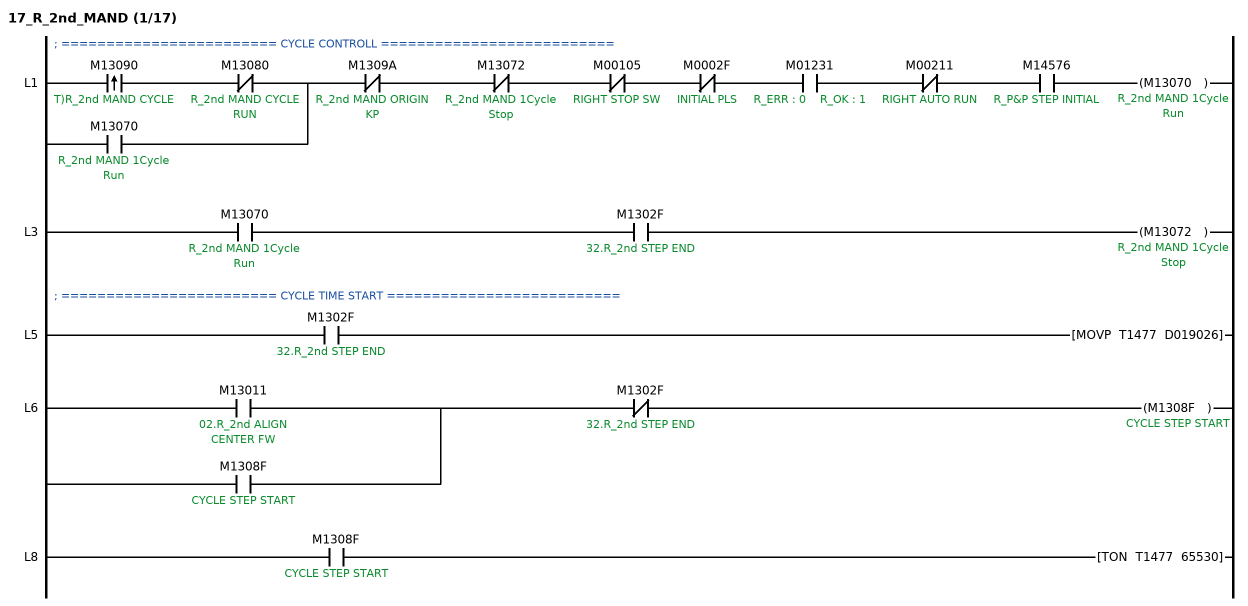
[picture p144: 17_R_2nd_MAND rungs L1-L8]
// ======================== CYCLE CONTROLL ==========================
; L1
LOADP     M13090	// T)R_2nd MAND CYCLE
AND NOT   M13080	// R_2nd MAND CYCLE RUN
OR        M13070	// R_2nd MAND 1Cycle Run
AND NOT   M1309A	// R_2nd MAND ORIGIN KP
AND NOT   M13072	// R_2nd MAND 1Cycle Stop
AND NOT   M00105	// RIGHT STOP SW
AND NOT   M0002F	// INITIAL PLS
AND       M01231	// R_ERR : 0    R_OK : 1
AND NOT   M00211	// RIGHT AUTO RUN
AND       M14576	// R_P&P STEP INITIAL
OUT       M13070	// R_2nd MAND 1Cycle Run
; L3
LOAD      M13070	// R_2nd MAND 1Cycle Run
AND       M1302F	// 32.R_2nd STEP END
OUT       M13072	// R_2nd MAND 1Cycle Stop
// ======================== CYCLE TIME START ==========================
; L5
LOAD      M1302F	// 32.R_2nd STEP END
MOVP      T1477 D019026
; L6
LOAD      M13011	// 02.R_2nd ALIGN CENTER FW
OR        M1308F	// CYCLE STEP START
AND NOT   M1302F	// 32.R_2nd STEP END
OUT       M1308F	// CYCLE STEP START
; L8
LOAD      M1308F	// CYCLE STEP START
TON       T1477 65530

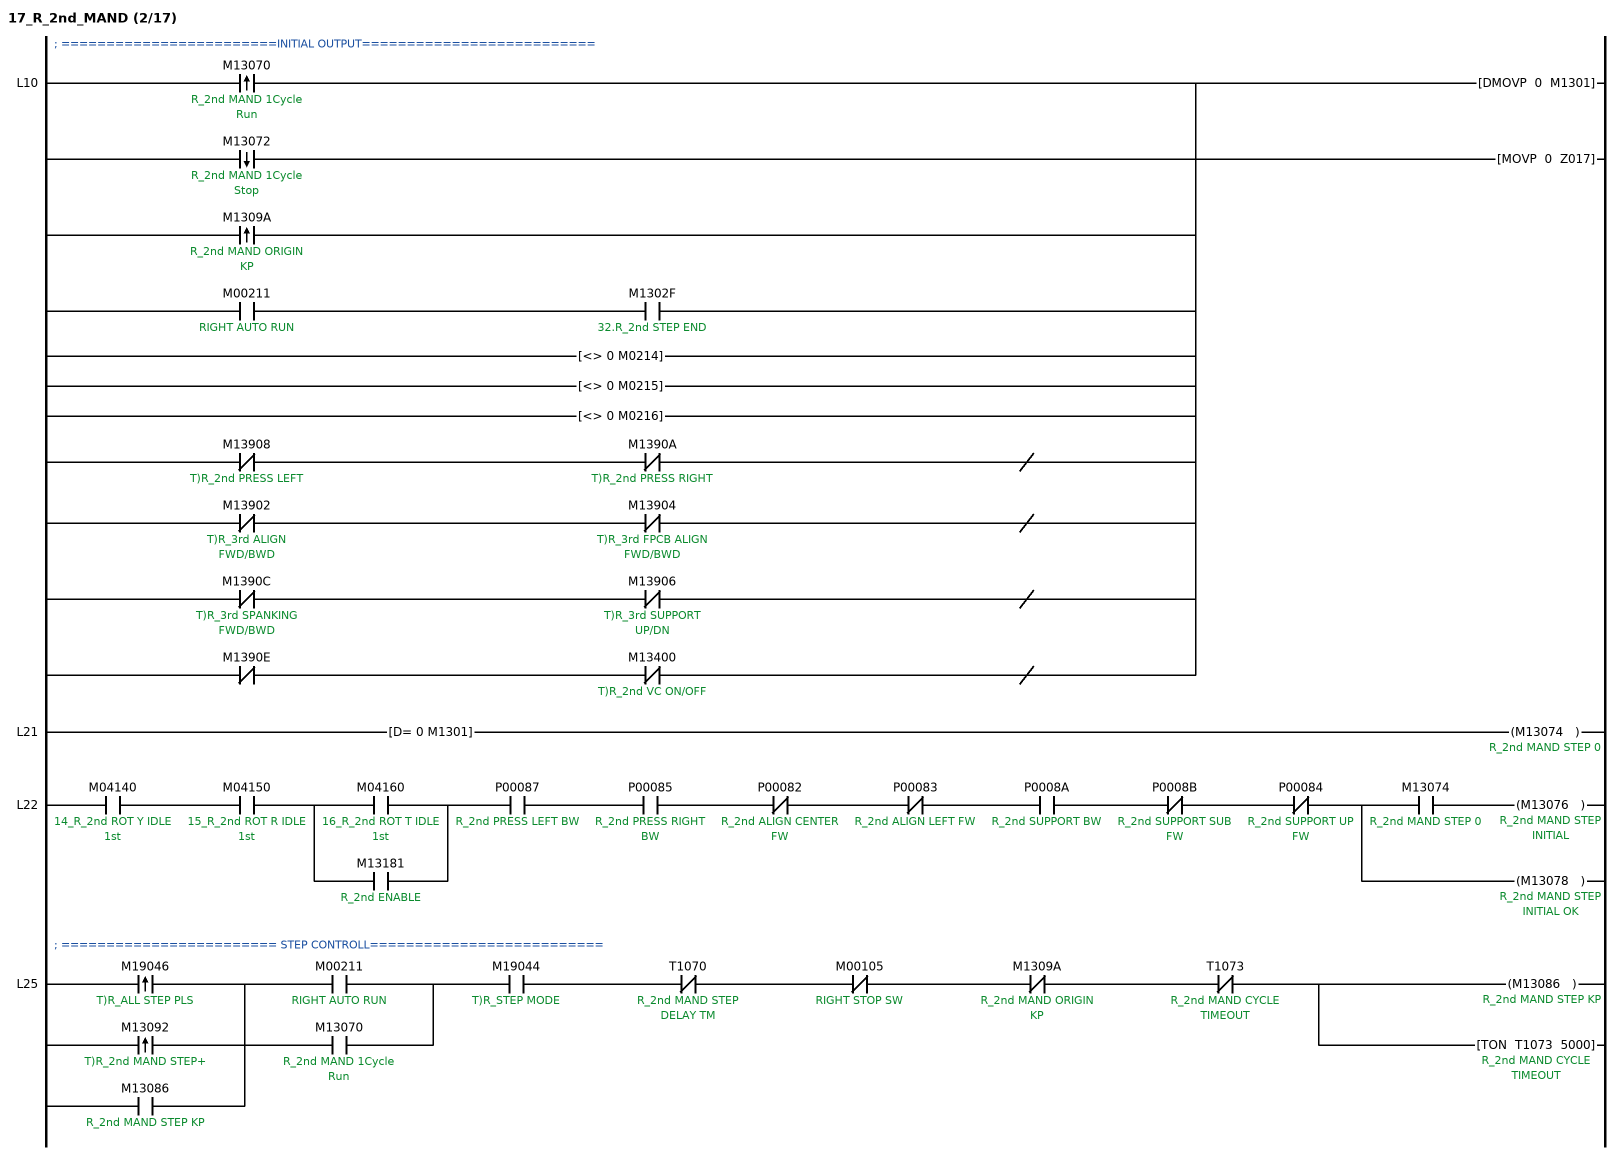
// ========================INITIAL OUTPUT==========================
; L10
LOADP     M13070	// R_2nd MAND 1Cycle Run
ORN       M13072	// R_2nd MAND 1Cycle Stop
ORP       M1309A	// R_2nd MAND ORIGIN KP
LOAD      M00211	// RIGHT AUTO RUN
AND       M1302F	// 32.R_2nd STEP END
OR LOAD
OR<>      0 M0214
OR<>      0 M0215
OR<>      0 M0216
LOAD NOT  M13908	// T)R_2nd PRESS LEFT
AND NOT   M1390A	// T)R_2nd PRESS RIGHT
NOT
OR LOAD
LOAD NOT  M13902	// T)R_3rd ALIGN FWD/BWD
AND NOT   M13904	// T)R_3rd FPCB ALIGN FWD/BWD
NOT
OR LOAD
LOAD NOT  M1390C	// T)R_3rd SPANKING FWD/BWD
AND NOT   M13906	// T)R_3rd SUPPORT UP/DN
NOT
OR LOAD
LOAD NOT  M1390E
AND NOT   M13400	// T)R_2nd VC ON/OFF
NOT
OR LOAD
DMOVP     0 M1301
MOVP      0 Z017
; L21
LOADD=    0 M1301
OUT       M13074	// R_2nd MAND STEP 0
; L22
LOAD      M04140	// 14_R_2nd ROT Y IDLE 1st
AND       M04150	// 15_R_2nd ROT R IDLE 1st
LOAD      M04160	// 16_R_2nd ROT T IDLE 1st
OR        M13181	// R_2nd ENABLE
AND LOAD
AND       P00087	// R_2nd PRESS LEFT BW
AND       P00085	// R_2nd PRESS RIGHT BW
AND NOT   P00082	// R_2nd ALIGN CENTER FW
AND NOT   P00083	// R_2nd ALIGN LEFT FW
AND       P0008A	// R_2nd SUPPORT BW
AND NOT   P0008B	// R_2nd SUPPORT SUB FW
AND NOT   P00084	// R_2nd SUPPORT UP FW
MPUSH
AND       M13074	// R_2nd MAND STEP 0
OUT       M13076	// R_2nd MAND STEP INITIAL
MPOP
OUT       M13078	// R_2nd MAND STEP INITIAL OK
// ======================== STEP CONTROLL==========================
; L25
LOADP     M19046	// T)R_ALL STEP PLS
ORP       M13092	// T)R_2nd MAND STEP+
OR        M13086	// R_2nd MAND STEP KP
LOAD      M00211	// RIGHT AUTO RUN
OR        M13070	// R_2nd MAND 1Cycle Run
AND LOAD
AND       M19044	// T)R_STEP MODE
AND NOT   T1070	// R_2nd MAND STEP DELAY TM
AND NOT   M00105	// RIGHT STOP SW
AND NOT   M1309A	// R_2nd MAND ORIGIN KP
AND NOT   T1073	// R_2nd MAND CYCLE TIMEOUT
OUT       M13086	// R_2nd MAND STEP KP
TON       T1073 5000	// R_2nd MAND CYCLE TIMEOUT

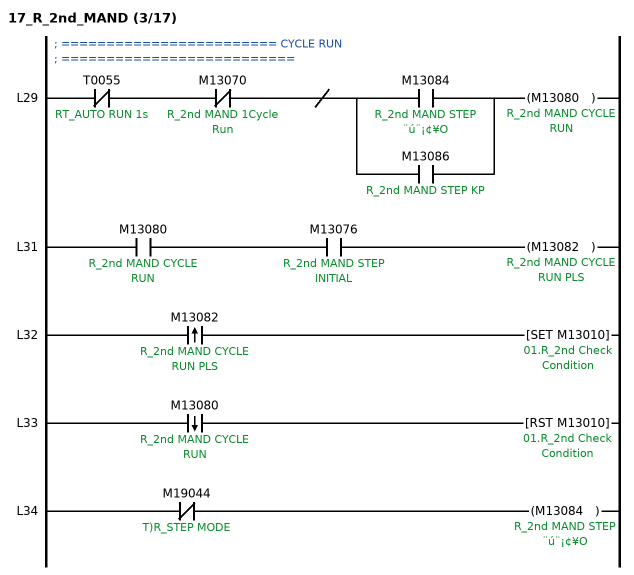
// ======================== CYCLE RUN ==========================
; L29
LOAD NOT  T0055	// RT_AUTO RUN 1s
AND NOT   M13070	// R_2nd MAND 1Cycle Run
NOT
LOAD      M13084	// R_2nd MAND STEP ¨ú¨¡¢¥O
OR        M13086	// R_2nd MAND STEP KP
AND LOAD
OUT       M13080	// R_2nd MAND CYCLE RUN
; L31
LOAD      M13080	// R_2nd MAND CYCLE RUN
AND       M13076	// R_2nd MAND STEP INITIAL
OUT       M13082	// R_2nd MAND CYCLE RUN PLS
; L32
LOADP     M13082	// R_2nd MAND CYCLE RUN PLS
SET       M13010	// 01.R_2nd Check Condition
; L33
LOADN     M13080	// R_2nd MAND CYCLE RUN
RST       M13010	// 01.R_2nd Check Condition
; L34
LOAD NOT  M19044	// T)R_STEP MODE
OUT       M13084	// R_2nd MAND STEP ¨ú¨¡¢¥O

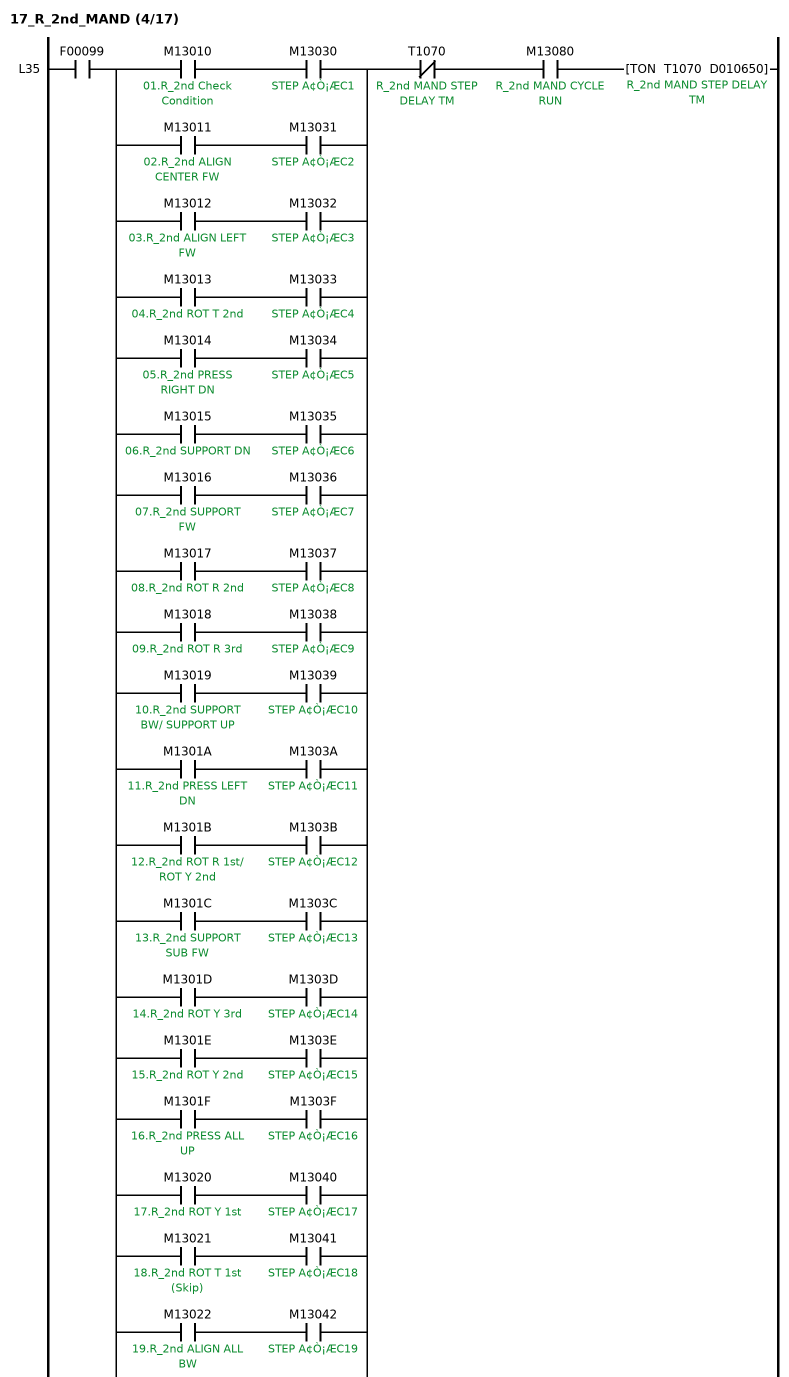

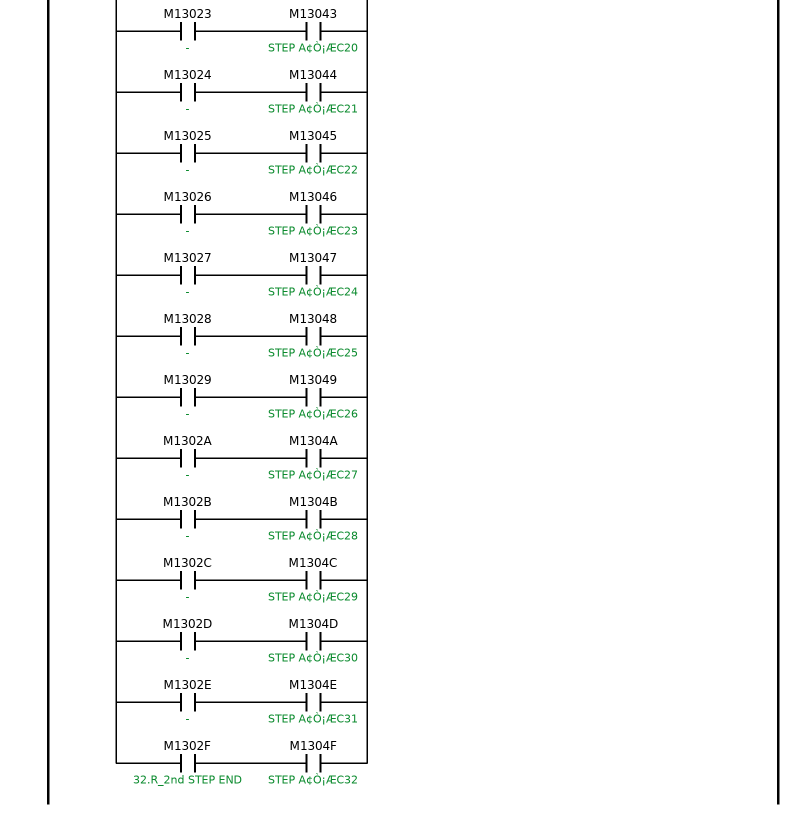
; L35
LOAD      F00099
LOAD      M13010	// 01.R_2nd Check Condition
AND       M13030	// STEP A¢Ò¡ÆC1
LOAD      M13011	// 02.R_2nd ALIGN CENTER FW
AND       M13031	// STEP A¢Ò¡ÆC2
OR LOAD
LOAD      M13012	// 03.R_2nd ALIGN LEFT FW
AND       M13032	// STEP A¢Ò¡ÆC3
OR LOAD
LOAD      M13013	// 04.R_2nd ROT T 2nd
AND       M13033	// STEP A¢Ò¡ÆC4
OR LOAD
LOAD      M13014	// 05.R_2nd PRESS RIGHT DN
AND       M13034	// STEP A¢Ò¡ÆC5
OR LOAD
LOAD      M13015	// 06.R_2nd SUPPORT DN
AND       M13035	// STEP A¢Ò¡ÆC6
OR LOAD
LOAD      M13016	// 07.R_2nd SUPPORT FW
AND       M13036	// STEP A¢Ò¡ÆC7
OR LOAD
LOAD      M13017	// 08.R_2nd ROT R 2nd
AND       M13037	// STEP A¢Ò¡ÆC8
OR LOAD
LOAD      M13018	// 09.R_2nd ROT R 3rd
AND       M13038	// STEP A¢Ò¡ÆC9
OR LOAD
LOAD      M13019	// 10.R_2nd SUPPORT BW/ SUPPORT UP
AND       M13039	// STEP A¢Ò¡ÆC10
OR LOAD
LOAD      M1301A	// 11.R_2nd PRESS LEFT DN
AND       M1303A	// STEP A¢Ò¡ÆC11
OR LOAD
LOAD      M1301B	// 12.R_2nd ROT R 1st/ ROT Y 2nd
AND       M1303B	// STEP A¢Ò¡ÆC12
OR LOAD
LOAD      M1301C	// 13.R_2nd SUPPORT SUB FW
AND       M1303C	// STEP A¢Ò¡ÆC13
OR LOAD
LOAD      M1301D	// 14.R_2nd ROT Y 3rd
AND       M1303D	// STEP A¢Ò¡ÆC14
OR LOAD
LOAD      M1301E	// 15.R_2nd ROT Y 2nd
AND       M1303E	// STEP A¢Ò¡ÆC15
OR LOAD
LOAD      M1301F	// 16.R_2nd PRESS ALL UP
AND       M1303F	// STEP A¢Ò¡ÆC16
OR LOAD
LOAD      M13020	// 17.R_2nd ROT Y 1st
AND       M13040	// STEP A¢Ò¡ÆC17
OR LOAD
LOAD      M13021	// 18.R_2nd ROT T 1st (Skip)
AND       M13041	// STEP A¢Ò¡ÆC18
OR LOAD
LOAD      M13022	// 19.R_2nd ALIGN ALL BW
AND       M13042	// STEP A¢Ò¡ÆC19
OR LOAD
LOAD      M13023	// -
AND       M13043	// STEP A¢Ò¡ÆC20
OR LOAD
LOAD      M13024	// -
AND       M13044	// STEP A¢Ò¡ÆC21
OR LOAD
LOAD      M13025	// -
AND       M13045	// STEP A¢Ò¡ÆC22
OR LOAD
LOAD      M13026	// -
AND       M13046	// STEP A¢Ò¡ÆC23
OR LOAD
LOAD      M13027	// -
AND       M13047	// STEP A¢Ò¡ÆC24
OR LOAD
LOAD      M13028	// -
AND       M13048	// STEP A¢Ò¡ÆC25
OR LOAD
LOAD      M13029	// -
AND       M13049	// STEP A¢Ò¡ÆC26
OR LOAD
LOAD      M1302A	// -
AND       M1304A	// STEP A¢Ò¡ÆC27
OR LOAD
LOAD      M1302B	// -
AND       M1304B	// STEP A¢Ò¡ÆC28
OR LOAD
LOAD      M1302C	// -
AND       M1304C	// STEP A¢Ò¡ÆC29
OR LOAD
LOAD      M1302D	// -
AND       M1304D	// STEP A¢Ò¡ÆC30
OR LOAD
LOAD      M1302E	// -
AND       M1304E	// STEP A¢Ò¡ÆC31
OR LOAD
LOAD      M1302F	// 32.R_2nd STEP END
AND       M1304F	// STEP A¢Ò¡ÆC32
OR LOAD
AND LOAD
AND NOT   T1070	// R_2nd MAND STEP DELAY TM
AND       M13080	// R_2nd MAND CYCLE RUN
TON       T1070 D010650	// R_2nd MAND STEP DELAY TM

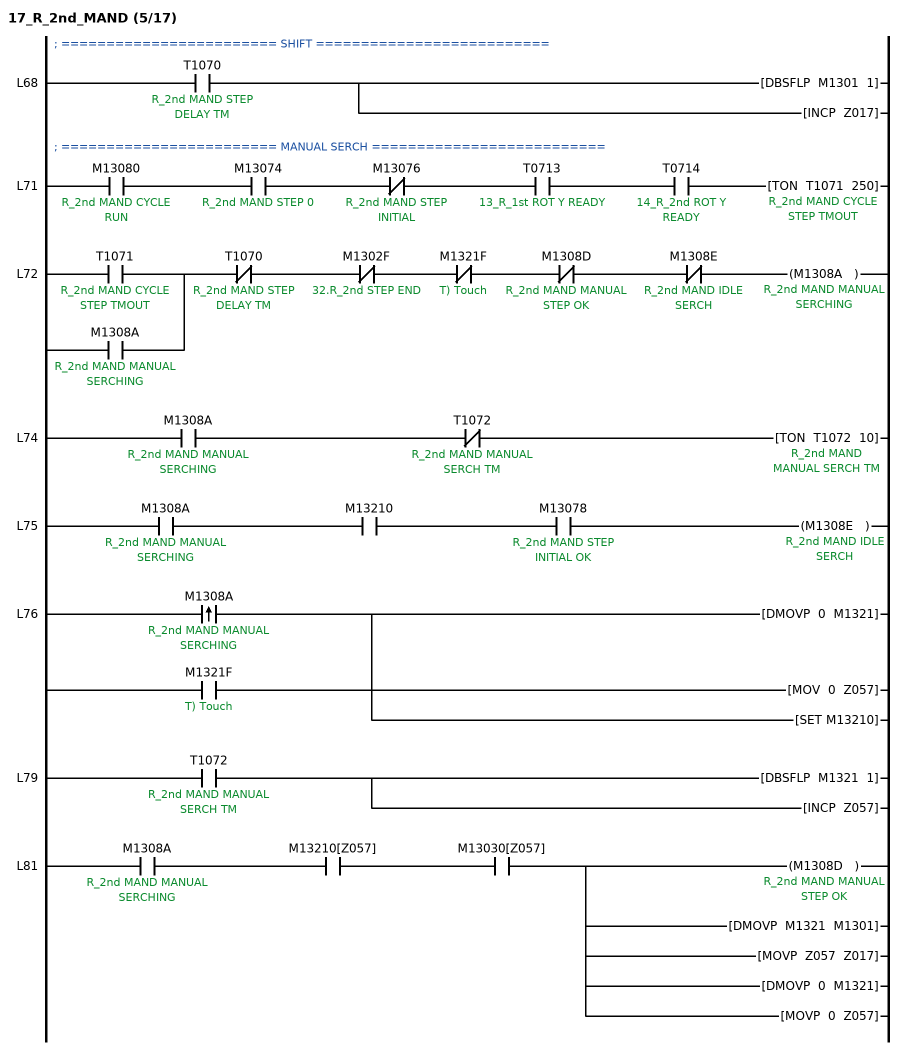
// ======================== SHIFT ==========================
; L68
LOAD      T1070	// R_2nd MAND STEP DELAY TM
DBSFLP    M1301 1
INCP      Z017
// ======================== MANUAL SERCH ==========================
; L71
LOAD      M13080	// R_2nd MAND CYCLE RUN
AND       M13074	// R_2nd MAND STEP 0
AND NOT   M13076	// R_2nd MAND STEP INITIAL
AND       T0713	// 13_R_1st ROT Y READY
AND       T0714	// 14_R_2nd ROT Y READY
TON       T1071 250	// R_2nd MAND CYCLE STEP TMOUT
; L72
LOAD      T1071	// R_2nd MAND CYCLE STEP TMOUT
OR        M1308A	// R_2nd MAND MANUAL SERCHING
AND NOT   T1070	// R_2nd MAND STEP DELAY TM
AND NOT   M1302F	// 32.R_2nd STEP END
AND NOT   M1321F	// T) Touch
AND NOT   M1308D	// R_2nd MAND MANUAL STEP OK
AND NOT   M1308E	// R_2nd MAND IDLE SERCH
OUT       M1308A	// R_2nd MAND MANUAL SERCHING
; L74
LOAD      M1308A	// R_2nd MAND MANUAL SERCHING
AND NOT   T1072	// R_2nd MAND MANUAL SERCH TM
TON       T1072 10	// R_2nd MAND MANUAL SERCH TM
; L75
LOAD      M1308A	// R_2nd MAND MANUAL SERCHING
AND       M13210
AND       M13078	// R_2nd MAND STEP INITIAL OK
OUT       M1308E	// R_2nd MAND IDLE SERCH
; L76
LOADP     M1308A	// R_2nd MAND MANUAL SERCHING
OR        M1321F	// T) Touch
DMOVP     0 M1321
MOV       0 Z057
SET       M13210
; L79
LOAD      T1072	// R_2nd MAND MANUAL SERCH TM
DBSFLP    M1321 1
INCP      Z057
; L81
LOAD      M1308A	// R_2nd MAND MANUAL SERCHING
AND       M13210[Z057]
AND       M13030[Z057]
OUT       M1308D	// R_2nd MAND MANUAL STEP OK
DMOVP     M1321 M1301
MOVP      Z057 Z017
DMOVP     0 M1321
MOVP      0 Z057

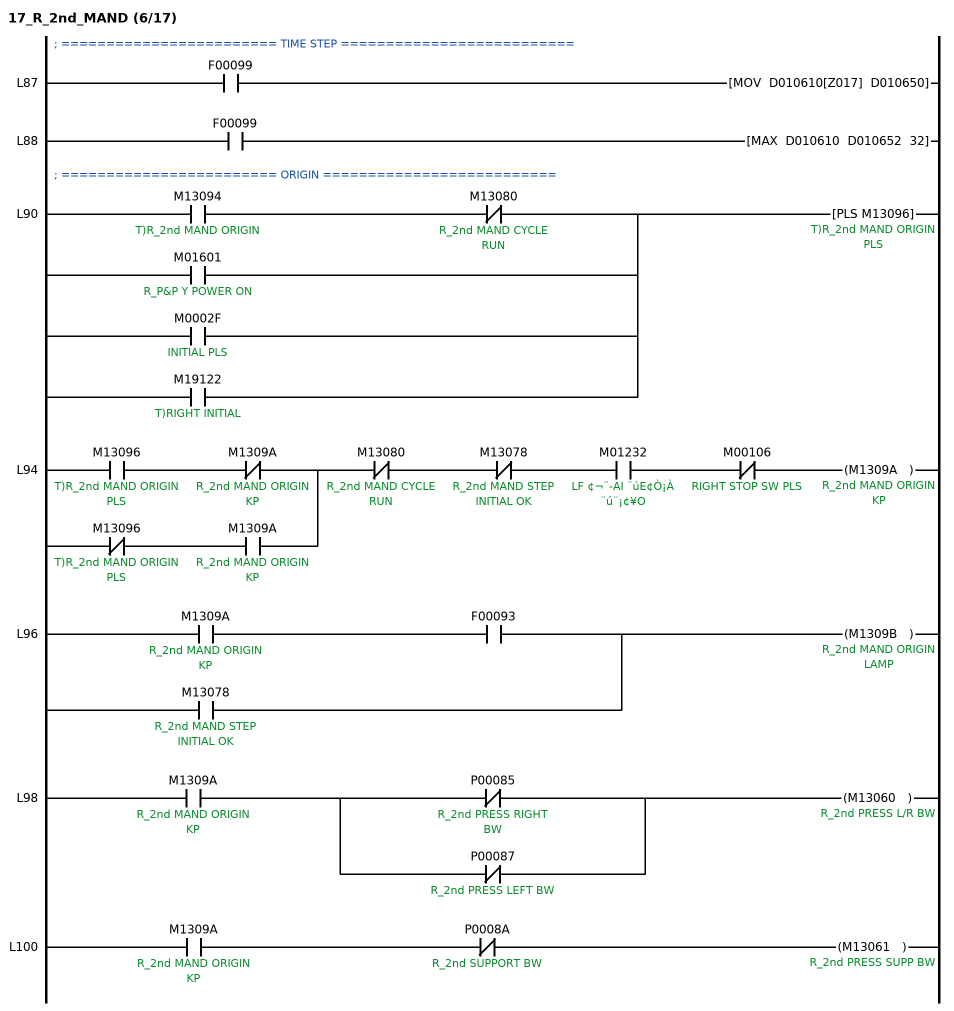
// ======================== TIME STEP ==========================
; L87
LOAD      F00099
MOV       D010610[Z017] D010650
; L88
LOAD      F00099
MAX       D010610 D010652 32
// ======================== ORIGIN ==========================
; L90
LOAD      M13094	// T)R_2nd MAND ORIGIN
AND NOT   M13080	// R_2nd MAND CYCLE RUN
OR        M01601	// R_P&P Y POWER ON
OR        M0002F	// INITIAL PLS
OR        M19122	// T)RIGHT INITIAL
OUTP      M13096	// T)R_2nd MAND ORIGIN PLS
; L94
LOAD      M13096	// T)R_2nd MAND ORIGIN PLS
AND NOT   M1309A	// R_2nd MAND ORIGIN KP
LOAD NOT  M13096	// T)R_2nd MAND ORIGIN PLS
AND       M1309A	// R_2nd MAND ORIGIN KP
OR LOAD
AND NOT   M13080	// R_2nd MAND CYCLE RUN
AND NOT   M13078	// R_2nd MAND STEP INITIAL OK
AND       M01232	// LF ¢¬¨­AI ¨úE¢Ò¡À ¨ú¨¡¢¥O
AND NOT   M00106	// RIGHT STOP SW PLS
OUT       M1309A	// R_2nd MAND ORIGIN KP
; L96
LOAD      M1309A	// R_2nd MAND ORIGIN KP
AND       F00093
OR        M13078	// R_2nd MAND STEP INITIAL OK
OUT       M1309B	// R_2nd MAND ORIGIN LAMP
; L98
LOAD      M1309A	// R_2nd MAND ORIGIN KP
LOAD NOT  P00085	// R_2nd PRESS RIGHT BW
OR NOT    P00087	// R_2nd PRESS LEFT BW
AND LOAD
OUT       M13060	// R_2nd PRESS L/R BW
; L100
LOAD      M1309A	// R_2nd MAND ORIGIN KP
AND NOT   P0008A	// R_2nd SUPPORT BW
OUT       M13061	// R_2nd PRESS SUPP BW

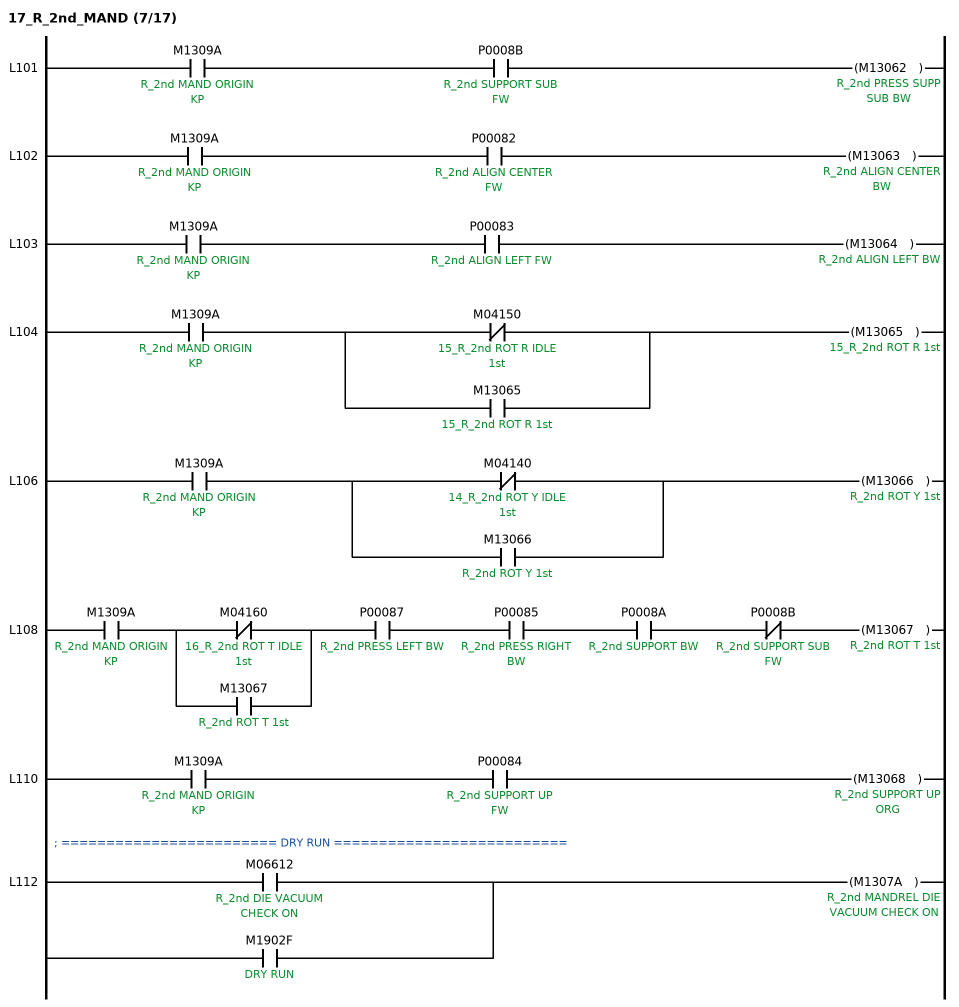
; L101
LOAD      M1309A	// R_2nd MAND ORIGIN KP
AND       P0008B	// R_2nd SUPPORT SUB FW
OUT       M13062	// R_2nd PRESS SUPP SUB BW
; L102
LOAD      M1309A	// R_2nd MAND ORIGIN KP
AND       P00082	// R_2nd ALIGN CENTER FW
OUT       M13063	// R_2nd ALIGN CENTER BW
; L103
LOAD      M1309A	// R_2nd MAND ORIGIN KP
AND       P00083	// R_2nd ALIGN LEFT FW
OUT       M13064	// R_2nd ALIGN LEFT BW
; L104
LOAD      M1309A	// R_2nd MAND ORIGIN KP
LOAD NOT  M04150	// 15_R_2nd ROT R IDLE 1st
OR        M13065	// 15_R_2nd ROT R 1st
AND LOAD
OUT       M13065	// 15_R_2nd ROT R 1st
; L106
LOAD      M1309A	// R_2nd MAND ORIGIN KP
LOAD NOT  M04140	// 14_R_2nd ROT Y IDLE 1st
OR        M13066	// R_2nd ROT Y 1st
AND LOAD
OUT       M13066	// R_2nd ROT Y 1st
; L108
LOAD      M1309A	// R_2nd MAND ORIGIN KP
LOAD NOT  M04160	// 16_R_2nd ROT T IDLE 1st
OR        M13067	// R_2nd ROT T 1st
AND LOAD
AND       P00087	// R_2nd PRESS LEFT BW
AND       P00085	// R_2nd PRESS RIGHT BW
AND       P0008A	// R_2nd SUPPORT BW
AND NOT   P0008B	// R_2nd SUPPORT SUB FW
OUT       M13067	// R_2nd ROT T 1st
; L110
LOAD      M1309A	// R_2nd MAND ORIGIN KP
AND       P00084	// R_2nd SUPPORT UP FW
OUT       M13068	// R_2nd SUPPORT UP ORG
// ======================== DRY RUN ==========================
; L112
LOAD      M06612	// R_2nd DIE VACUUM CHECK ON
OR        M1902F	// DRY RUN
OUT       M1307A	// R_2nd MANDREL DIE VACUUM CHECK ON

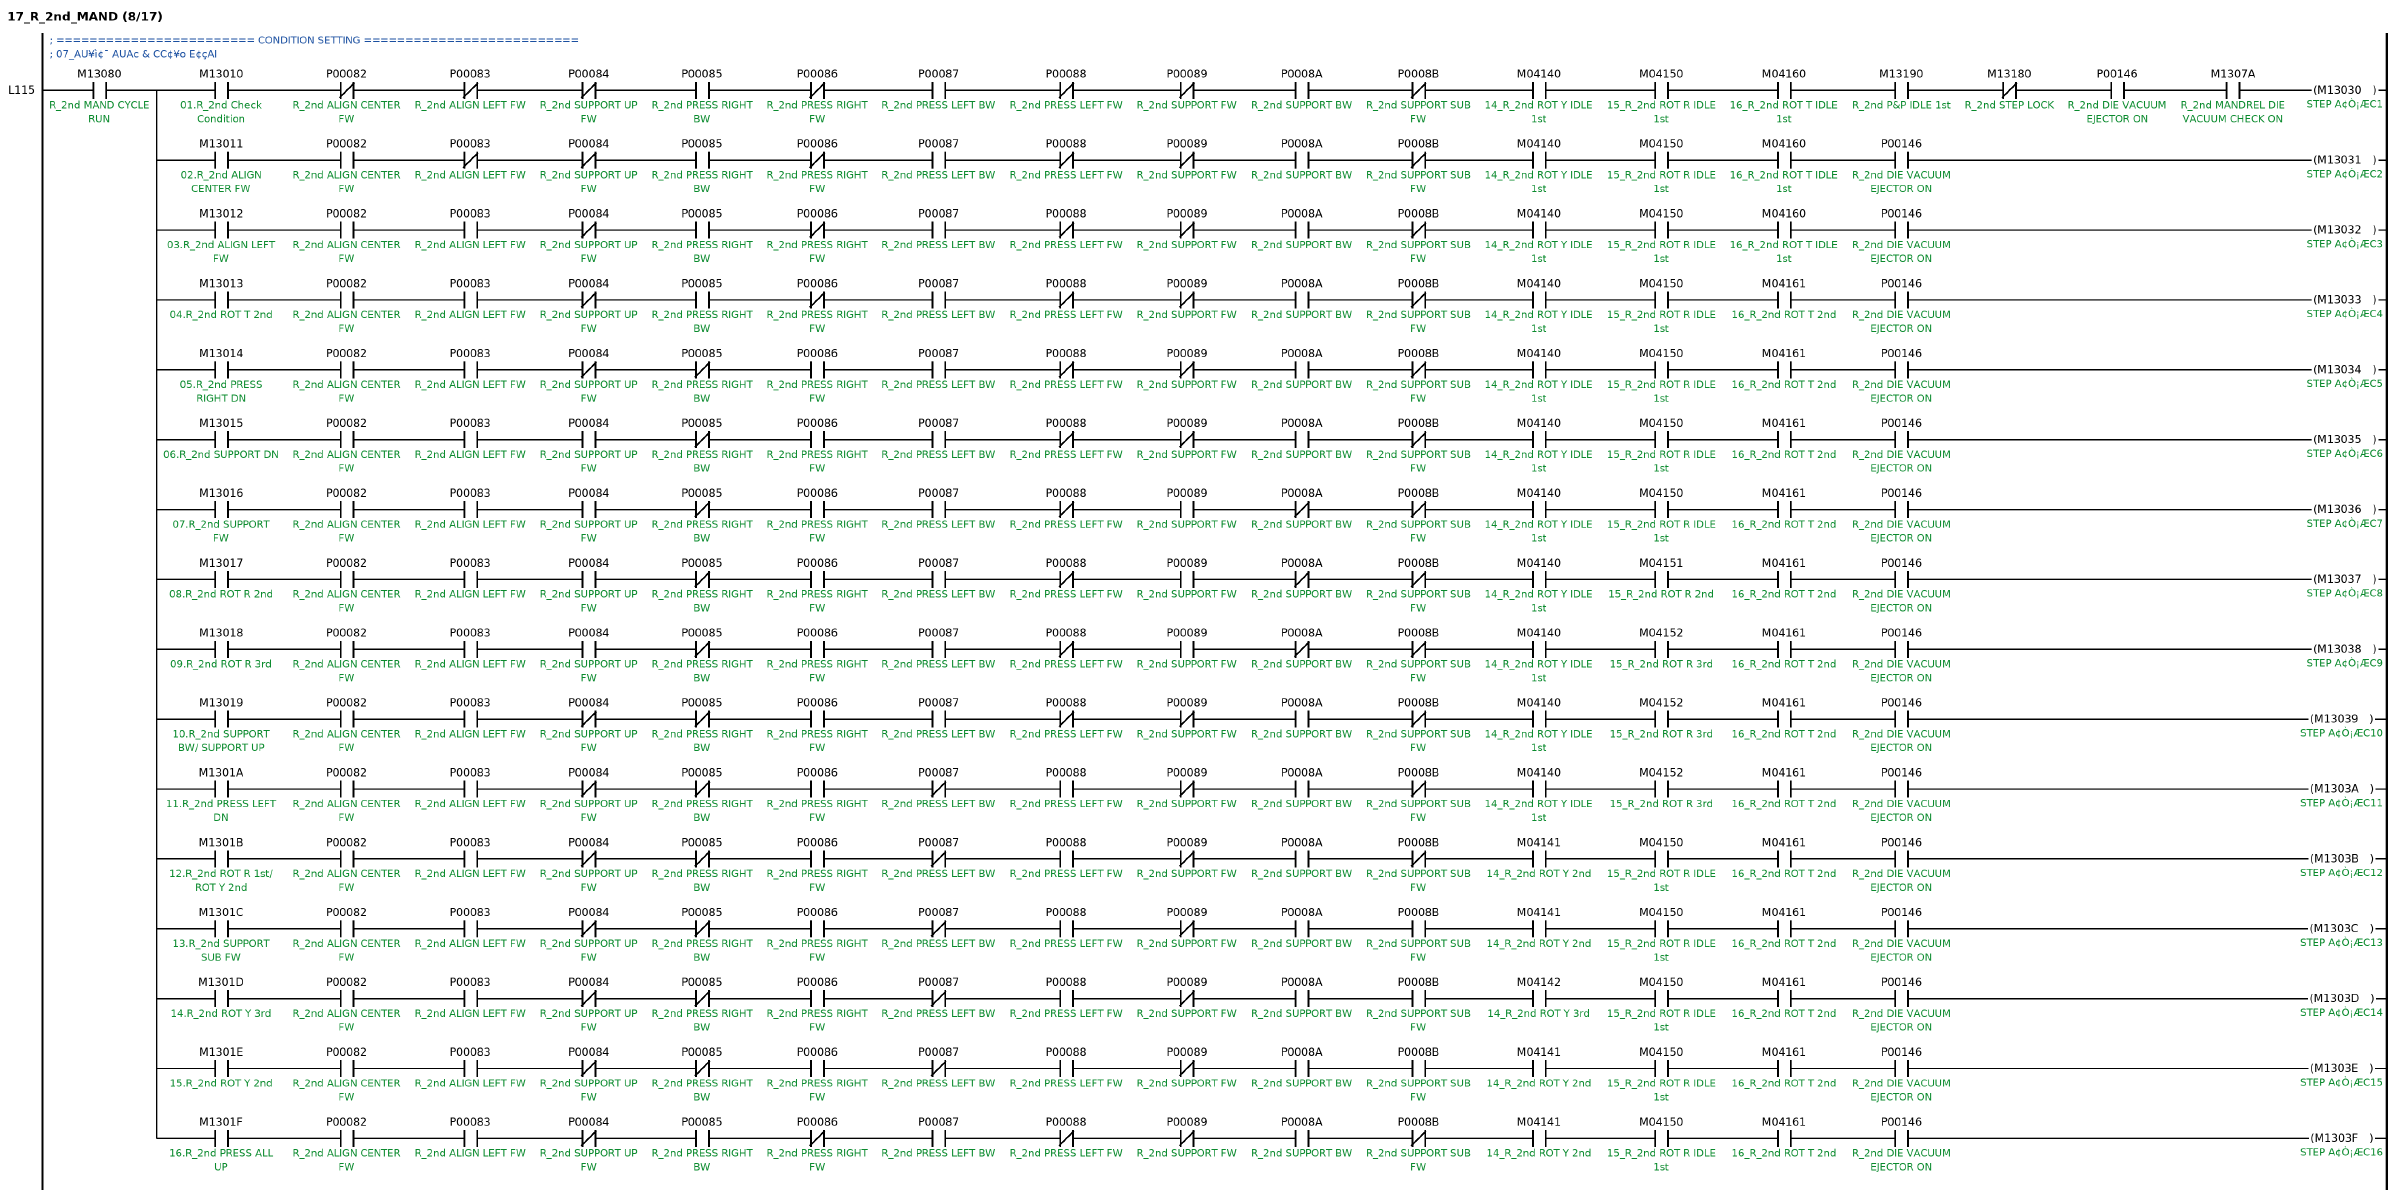
// ======================== CONDITION SETTING ==========================
; L115
LOAD      M13080	// R_2nd MAND CYCLE RUN
MPUSH
AND       M13010	// 01.R_2nd Check Condition
AND NOT   P00082	// R_2nd ALIGN CENTER FW
AND NOT   P00083	// R_2nd ALIGN LEFT FW
AND NOT   P00084	// R_2nd SUPPORT UP FW
AND       P00085	// R_2nd PRESS RIGHT BW
AND NOT   P00086	// R_2nd PRESS RIGHT FW
AND       P00087	// R_2nd PRESS LEFT BW
AND NOT   P00088	// R_2nd PRESS LEFT FW
AND NOT   P00089	// R_2nd SUPPORT FW
AND       P0008A	// R_2nd SUPPORT BW
AND NOT   P0008B	// R_2nd SUPPORT SUB FW
AND       M04140	// 14_R_2nd ROT Y IDLE 1st
AND       M04150	// 15_R_2nd ROT R IDLE 1st
AND       M04160	// 16_R_2nd ROT T IDLE 1st
AND       M13190	// R_2nd P&P IDLE 1st
AND NOT   M13180	// R_2nd STEP LOCK
AND       P00146	// R_2nd DIE VACUUM EJECTOR ON
AND       M1307A	// R_2nd MANDREL DIE VACUUM CHECK ON
OUT       M13030	// STEP A¢Ò¡ÆC1
MLOAD
AND       M13011	// 02.R_2nd ALIGN CENTER FW
AND       P00082	// R_2nd ALIGN CENTER FW
AND NOT   P00083	// R_2nd ALIGN LEFT FW
AND NOT   P00084	// R_2nd SUPPORT UP FW
AND       P00085	// R_2nd PRESS RIGHT BW
AND NOT   P00086	// R_2nd PRESS RIGHT FW
AND       P00087	// R_2nd PRESS LEFT BW
AND NOT   P00088	// R_2nd PRESS LEFT FW
AND NOT   P00089	// R_2nd SUPPORT FW
AND       P0008A	// R_2nd SUPPORT BW
AND NOT   P0008B	// R_2nd SUPPORT SUB FW
AND       M04140	// 14_R_2nd ROT Y IDLE 1st
AND       M04150	// 15_R_2nd ROT R IDLE 1st
AND       M04160	// 16_R_2nd ROT T IDLE 1st
AND       P00146	// R_2nd DIE VACUUM EJECTOR ON
OUT       M13031	// STEP A¢Ò¡ÆC2
MLOAD
AND       M13012	// 03.R_2nd ALIGN LEFT FW
AND       P00082	// R_2nd ALIGN CENTER FW
AND       P00083	// R_2nd ALIGN LEFT FW
AND NOT   P00084	// R_2nd SUPPORT UP FW
AND       P00085	// R_2nd PRESS RIGHT BW
AND NOT   P00086	// R_2nd PRESS RIGHT FW
AND       P00087	// R_2nd PRESS LEFT BW
AND NOT   P00088	// R_2nd PRESS LEFT FW
AND NOT   P00089	// R_2nd SUPPORT FW
AND       P0008A	// R_2nd SUPPORT BW
AND NOT   P0008B	// R_2nd SUPPORT SUB FW
AND       M04140	// 14_R_2nd ROT Y IDLE 1st
AND       M04150	// 15_R_2nd ROT R IDLE 1st
AND       M04160	// 16_R_2nd ROT T IDLE 1st
AND       P00146	// R_2nd DIE VACUUM EJECTOR ON
OUT       M13032	// STEP A¢Ò¡ÆC3
MLOAD
AND       M13013	// 04.R_2nd ROT T 2nd
AND       P00082	// R_2nd ALIGN CENTER FW
AND       P00083	// R_2nd ALIGN LEFT FW
AND NOT   P00084	// R_2nd SUPPORT UP FW
AND       P00085	// R_2nd PRESS RIGHT BW
AND NOT   P00086	// R_2nd PRESS RIGHT FW
AND       P00087	// R_2nd PRESS LEFT BW
AND NOT   P00088	// R_2nd PRESS LEFT FW
AND NOT   P00089	// R_2nd SUPPORT FW
AND       P0008A	// R_2nd SUPPORT BW
AND NOT   P0008B	// R_2nd SUPPORT SUB FW
AND       M04140	// 14_R_2nd ROT Y IDLE 1st
AND       M04150	// 15_R_2nd ROT R IDLE 1st
AND       M04161	// 16_R_2nd ROT T 2nd
AND       P00146	// R_2nd DIE VACUUM EJECTOR ON
OUT       M13033	// STEP A¢Ò¡ÆC4
MLOAD
AND       M13014	// 05.R_2nd PRESS RIGHT DN
AND       P00082	// R_2nd ALIGN CENTER FW
AND       P00083	// R_2nd ALIGN LEFT FW
AND NOT   P00084	// R_2nd SUPPORT UP FW
AND NOT   P00085	// R_2nd PRESS RIGHT BW
AND       P00086	// R_2nd PRESS RIGHT FW
AND       P00087	// R_2nd PRESS LEFT BW
AND NOT   P00088	// R_2nd PRESS LEFT FW
AND NOT   P00089	// R_2nd SUPPORT FW
AND       P0008A	// R_2nd SUPPORT BW
AND NOT   P0008B	// R_2nd SUPPORT SUB FW
AND       M04140	// 14_R_2nd ROT Y IDLE 1st
AND       M04150	// 15_R_2nd ROT R IDLE 1st
AND       M04161	// 16_R_2nd ROT T 2nd
AND       P00146	// R_2nd DIE VACUUM EJECTOR ON
OUT       M13034	// STEP A¢Ò¡ÆC5
MLOAD
AND       M13015	// 06.R_2nd SUPPORT DN
AND       P00082	// R_2nd ALIGN CENTER FW
AND       P00083	// R_2nd ALIGN LEFT FW
AND       P00084	// R_2nd SUPPORT UP FW
AND NOT   P00085	// R_2nd PRESS RIGHT BW
AND       P00086	// R_2nd PRESS RIGHT FW
AND       P00087	// R_2nd PRESS LEFT BW
AND NOT   P00088	// R_2nd PRESS LEFT FW
AND NOT   P00089	// R_2nd SUPPORT FW
AND       P0008A	// R_2nd SUPPORT BW
AND NOT   P0008B	// R_2nd SUPPORT SUB FW
AND       M04140	// 14_R_2nd ROT Y IDLE 1st
AND       M04150	// 15_R_2nd ROT R IDLE 1st
AND       M04161	// 16_R_2nd ROT T 2nd
AND       P00146	// R_2nd DIE VACUUM EJECTOR ON
OUT       M13035	// STEP A¢Ò¡ÆC6
MLOAD
AND       M13016	// 07.R_2nd SUPPORT FW
AND       P00082	// R_2nd ALIGN CENTER FW
AND       P00083	// R_2nd ALIGN LEFT FW
AND       P00084	// R_2nd SUPPORT UP FW
AND NOT   P00085	// R_2nd PRESS RIGHT BW
AND       P00086	// R_2nd PRESS RIGHT FW
AND       P00087	// R_2nd PRESS LEFT BW
AND NOT   P00088	// R_2nd PRESS LEFT FW
AND       P00089	// R_2nd SUPPORT FW
AND NOT   P0008A	// R_2nd SUPPORT BW
AND NOT   P0008B	// R_2nd SUPPORT SUB FW
AND       M04140	// 14_R_2nd ROT Y IDLE 1st
AND       M04150	// 15_R_2nd ROT R IDLE 1st
AND       M04161	// 16_R_2nd ROT T 2nd
AND       P00146	// R_2nd DIE VACUUM EJECTOR ON
OUT       M13036	// STEP A¢Ò¡ÆC7
MLOAD
AND       M13017	// 08.R_2nd ROT R 2nd
AND       P00082	// R_2nd ALIGN CENTER FW
AND       P00083	// R_2nd ALIGN LEFT FW
AND       P00084	// R_2nd SUPPORT UP FW
AND NOT   P00085	// R_2nd PRESS RIGHT BW
AND       P00086	// R_2nd PRESS RIGHT FW
AND       P00087	// R_2nd PRESS LEFT BW
AND NOT   P00088	// R_2nd PRESS LEFT FW
AND       P00089	// R_2nd SUPPORT FW
AND NOT   P0008A	// R_2nd SUPPORT BW
AND NOT   P0008B	// R_2nd SUPPORT SUB FW
AND       M04140	// 14_R_2nd ROT Y IDLE 1st
AND       M04151	// 15_R_2nd ROT R 2nd
AND       M04161	// 16_R_2nd ROT T 2nd
AND       P00146	// R_2nd DIE VACUUM EJECTOR ON
OUT       M13037	// STEP A¢Ò¡ÆC8
MLOAD
AND       M13018	// 09.R_2nd ROT R 3rd
AND       P00082	// R_2nd ALIGN CENTER FW
AND       P00083	// R_2nd ALIGN LEFT FW
AND       P00084	// R_2nd SUPPORT UP FW
AND NOT   P00085	// R_2nd PRESS RIGHT BW
AND       P00086	// R_2nd PRESS RIGHT FW
AND       P00087	// R_2nd PRESS LEFT BW
AND NOT   P00088	// R_2nd PRESS LEFT FW
AND       P00089	// R_2nd SUPPORT FW
AND NOT   P0008A	// R_2nd SUPPORT BW
AND NOT   P0008B	// R_2nd SUPPORT SUB FW
AND       M04140	// 14_R_2nd ROT Y IDLE 1st
AND       M04152	// 15_R_2nd ROT R 3rd
AND       M04161	// 16_R_2nd ROT T 2nd
AND       P00146	// R_2nd DIE VACUUM EJECTOR ON
OUT       M13038	// STEP A¢Ò¡ÆC9
MLOAD
AND       M13019	// 10.R_2nd SUPPORT BW/ SUPPORT UP
AND       P00082	// R_2nd ALIGN CENTER FW
AND       P00083	// R_2nd ALIGN LEFT FW
AND NOT   P00084	// R_2nd SUPPORT UP FW
AND NOT   P00085	// R_2nd PRESS RIGHT BW
AND       P00086	// R_2nd PRESS RIGHT FW
AND       P00087	// R_2nd PRESS LEFT BW
AND NOT   P00088	// R_2nd PRESS LEFT FW
AND NOT   P00089	// R_2nd SUPPORT FW
AND       P0008A	// R_2nd SUPPORT BW
AND NOT   P0008B	// R_2nd SUPPORT SUB FW
AND       M04140	// 14_R_2nd ROT Y IDLE 1st
AND       M04152	// 15_R_2nd ROT R 3rd
AND       M04161	// 16_R_2nd ROT T 2nd
AND       P00146	// R_2nd DIE VACUUM EJECTOR ON
OUT       M13039	// STEP A¢Ò¡ÆC10
MLOAD
AND       M1301A	// 11.R_2nd PRESS LEFT DN
AND       P00082	// R_2nd ALIGN CENTER FW
AND       P00083	// R_2nd ALIGN LEFT FW
AND NOT   P00084	// R_2nd SUPPORT UP FW
AND NOT   P00085	// R_2nd PRESS RIGHT BW
AND       P00086	// R_2nd PRESS RIGHT FW
AND NOT   P00087	// R_2nd PRESS LEFT BW
AND       P00088	// R_2nd PRESS LEFT FW
AND NOT   P00089	// R_2nd SUPPORT FW
AND       P0008A	// R_2nd SUPPORT BW
AND NOT   P0008B	// R_2nd SUPPORT SUB FW
AND       M04140	// 14_R_2nd ROT Y IDLE 1st
AND       M04152	// 15_R_2nd ROT R 3rd
AND       M04161	// 16_R_2nd ROT T 2nd
AND       P00146	// R_2nd DIE VACUUM EJECTOR ON
OUT       M1303A	// STEP A¢Ò¡ÆC11
MLOAD
AND       M1301B	// 12.R_2nd ROT R 1st/ ROT Y 2nd
AND       P00082	// R_2nd ALIGN CENTER FW
AND       P00083	// R_2nd ALIGN LEFT FW
AND NOT   P00084	// R_2nd SUPPORT UP FW
AND NOT   P00085	// R_2nd PRESS RIGHT BW
AND       P00086	// R_2nd PRESS RIGHT FW
AND NOT   P00087	// R_2nd PRESS LEFT BW
AND       P00088	// R_2nd PRESS LEFT FW
AND NOT   P00089	// R_2nd SUPPORT FW
AND       P0008A	// R_2nd SUPPORT BW
AND NOT   P0008B	// R_2nd SUPPORT SUB FW
AND       M04141	// 14_R_2nd ROT Y 2nd
AND       M04150	// 15_R_2nd ROT R IDLE 1st
AND       M04161	// 16_R_2nd ROT T 2nd
AND       P00146	// R_2nd DIE VACUUM EJECTOR ON
OUT       M1303B	// STEP A¢Ò¡ÆC12
MLOAD
AND       M1301C	// 13.R_2nd SUPPORT SUB FW
AND       P00082	// R_2nd ALIGN CENTER FW
AND       P00083	// R_2nd ALIGN LEFT FW
AND NOT   P00084	// R_2nd SUPPORT UP FW
AND NOT   P00085	// R_2nd PRESS RIGHT BW
AND       P00086	// R_2nd PRESS RIGHT FW
AND NOT   P00087	// R_2nd PRESS LEFT BW
AND       P00088	// R_2nd PRESS LEFT FW
AND NOT   P00089	// R_2nd SUPPORT FW
AND       P0008A	// R_2nd SUPPORT BW
AND       P0008B	// R_2nd SUPPORT SUB FW
AND       M04141	// 14_R_2nd ROT Y 2nd
AND       M04150	// 15_R_2nd ROT R IDLE 1st
AND       M04161	// 16_R_2nd ROT T 2nd
AND       P00146	// R_2nd DIE VACUUM EJECTOR ON
OUT       M1303C	// STEP A¢Ò¡ÆC13
MLOAD
AND       M1301D	// 14.R_2nd ROT Y 3rd
AND       P00082	// R_2nd ALIGN CENTER FW
AND       P00083	// R_2nd ALIGN LEFT FW
AND NOT   P00084	// R_2nd SUPPORT UP FW
AND NOT   P00085	// R_2nd PRESS RIGHT BW
AND       P00086	// R_2nd PRESS RIGHT FW
AND NOT   P00087	// R_2nd PRESS LEFT BW
AND       P00088	// R_2nd PRESS LEFT FW
AND NOT   P00089	// R_2nd SUPPORT FW
AND       P0008A	// R_2nd SUPPORT BW
AND       P0008B	// R_2nd SUPPORT SUB FW
AND       M04142	// 14_R_2nd ROT Y 3rd
AND       M04150	// 15_R_2nd ROT R IDLE 1st
AND       M04161	// 16_R_2nd ROT T 2nd
AND       P00146	// R_2nd DIE VACUUM EJECTOR ON
OUT       M1303D	// STEP A¢Ò¡ÆC14
MLOAD
AND       M1301E	// 15.R_2nd ROT Y 2nd
AND       P00082	// R_2nd ALIGN CENTER FW
AND       P00083	// R_2nd ALIGN LEFT FW
AND NOT   P00084	// R_2nd SUPPORT UP FW
AND NOT   P00085	// R_2nd PRESS RIGHT BW
AND       P00086	// R_2nd PRESS RIGHT FW
AND NOT   P00087	// R_2nd PRESS LEFT BW
AND       P00088	// R_2nd PRESS LEFT FW
AND NOT   P00089	// R_2nd SUPPORT FW
AND       P0008A	// R_2nd SUPPORT BW
AND       P0008B	// R_2nd SUPPORT SUB FW
AND       M04141	// 14_R_2nd ROT Y 2nd
AND       M04150	// 15_R_2nd ROT R IDLE 1st
AND       M04161	// 16_R_2nd ROT T 2nd
AND       P00146	// R_2nd DIE VACUUM EJECTOR ON
OUT       M1303E	// STEP A¢Ò¡ÆC15
MPOP
AND       M1301F	// 16.R_2nd PRESS ALL UP
AND       P00082	// R_2nd ALIGN CENTER FW
AND       P00083	// R_2nd ALIGN LEFT FW
AND NOT   P00084	// R_2nd SUPPORT UP FW
AND       P00085	// R_2nd PRESS RIGHT BW
AND NOT   P00086	// R_2nd PRESS RIGHT FW
AND       P00087	// R_2nd PRESS LEFT BW
AND NOT   P00088	// R_2nd PRESS LEFT FW
AND NOT   P00089	// R_2nd SUPPORT FW
AND       P0008A	// R_2nd SUPPORT BW
AND NOT   P0008B	// R_2nd SUPPORT SUB FW
AND       M04141	// 14_R_2nd ROT Y 2nd
AND       M04150	// 15_R_2nd ROT R IDLE 1st
AND       M04161	// 16_R_2nd ROT T 2nd
AND       P00146	// R_2nd DIE VACUUM EJECTOR ON
OUT       M1303F	// STEP A¢Ò¡ÆC16
// output comment: 07_AU¥ì¢¯ AUAc & CC¢¥o E¢çAI

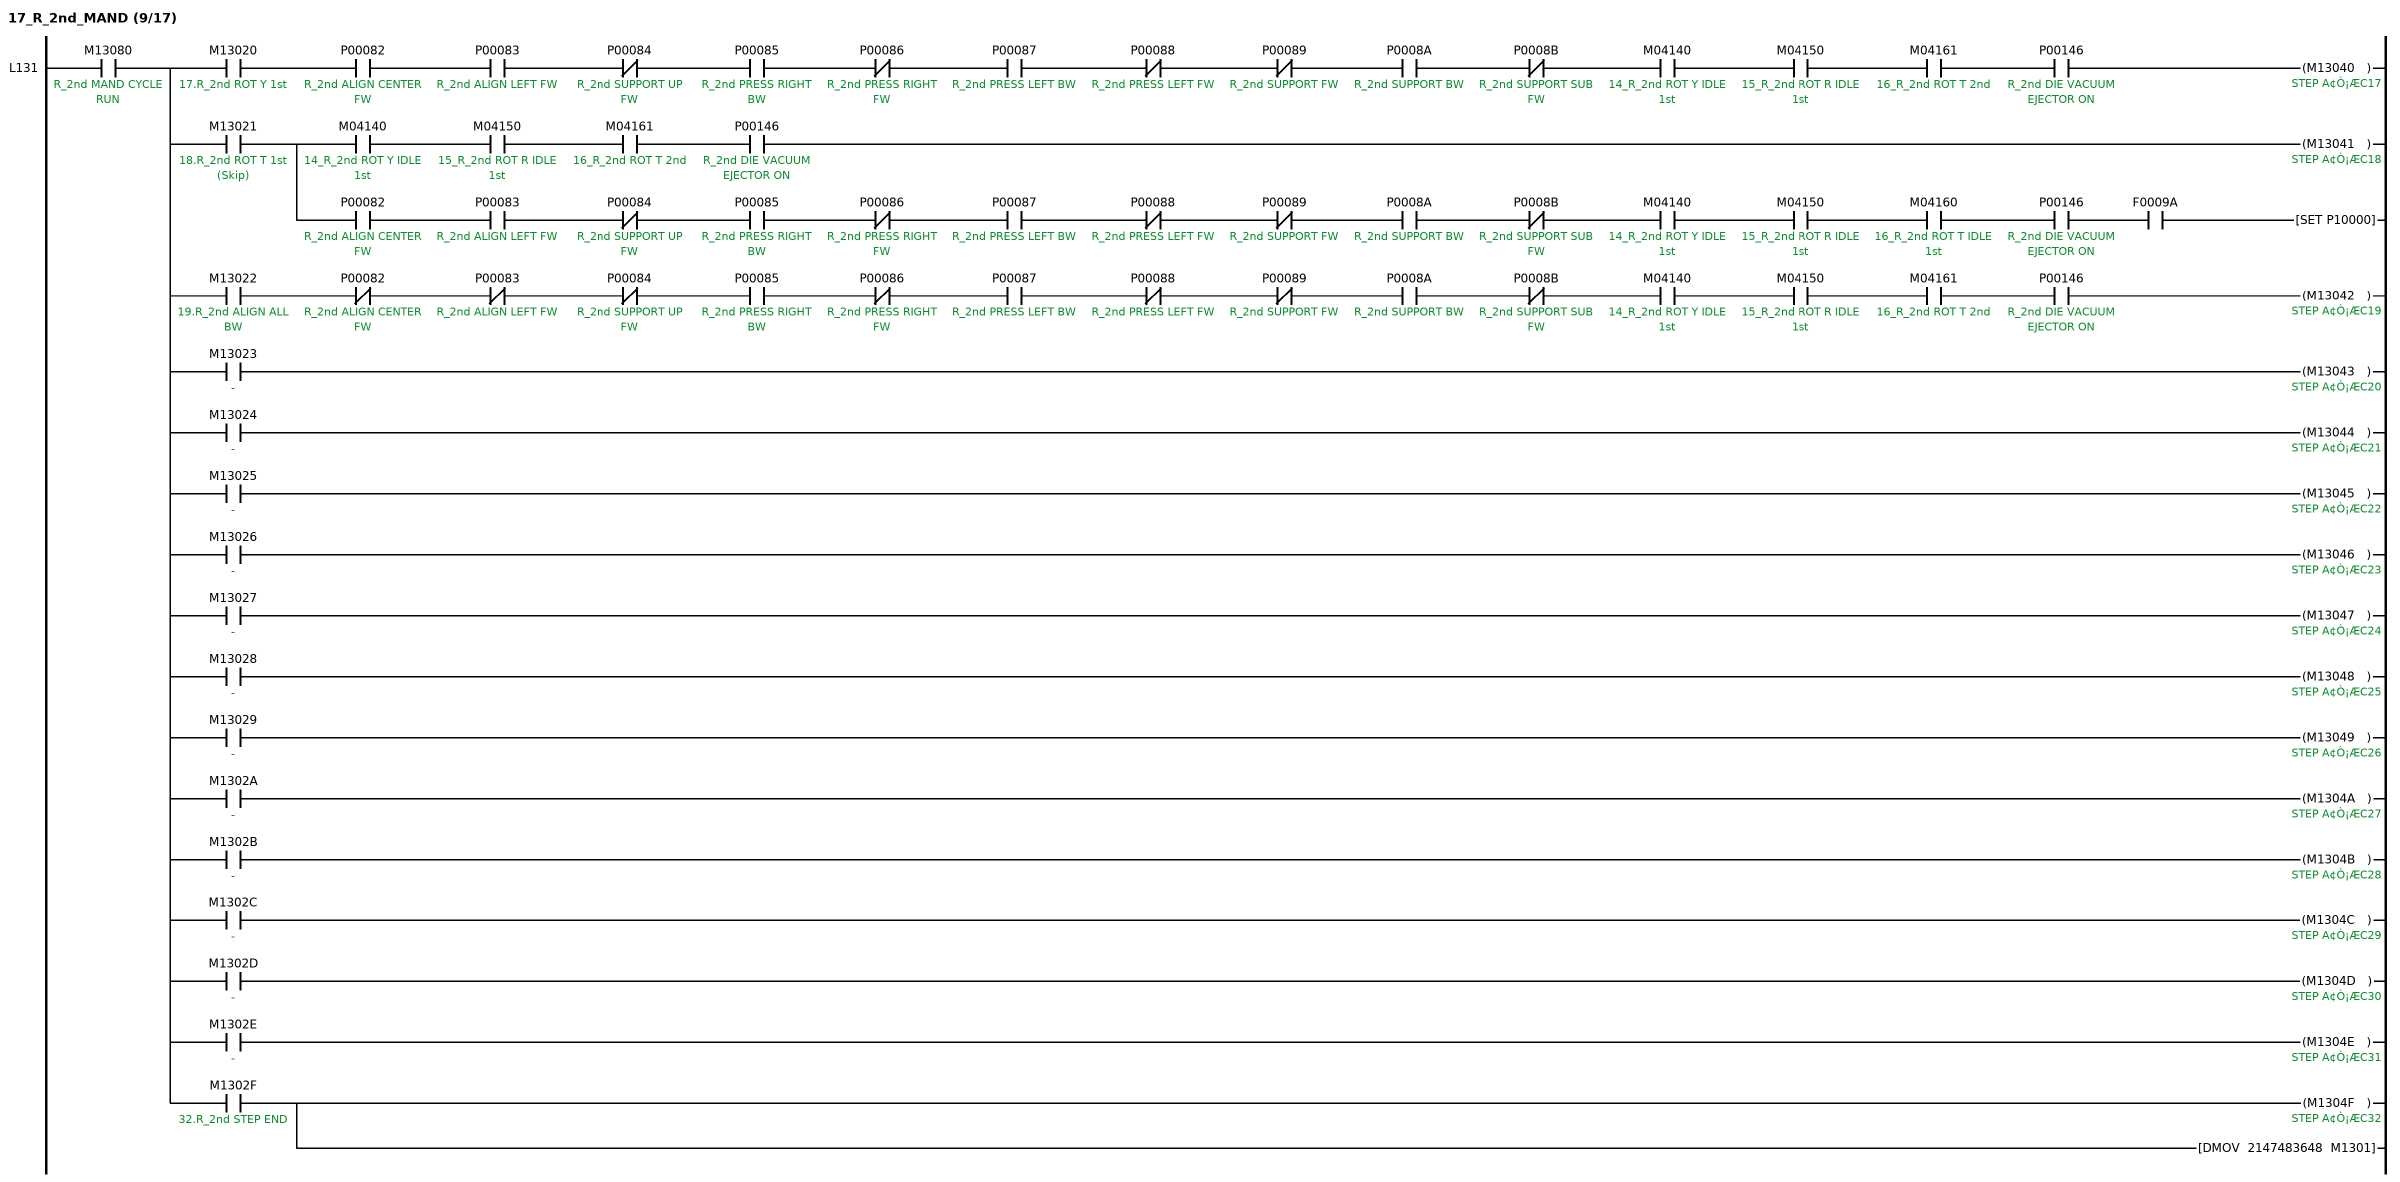
; L131
LOAD      M13080	// R_2nd MAND CYCLE RUN
MPUSH
AND       M13020	// 17.R_2nd ROT Y 1st
AND       P00082	// R_2nd ALIGN CENTER FW
AND       P00083	// R_2nd ALIGN LEFT FW
AND NOT   P00084	// R_2nd SUPPORT UP FW
AND       P00085	// R_2nd PRESS RIGHT BW
AND NOT   P00086	// R_2nd PRESS RIGHT FW
AND       P00087	// R_2nd PRESS LEFT BW
AND NOT   P00088	// R_2nd PRESS LEFT FW
AND NOT   P00089	// R_2nd SUPPORT FW
AND       P0008A	// R_2nd SUPPORT BW
AND NOT   P0008B	// R_2nd SUPPORT SUB FW
AND       M04140	// 14_R_2nd ROT Y IDLE 1st
AND       M04150	// 15_R_2nd ROT R IDLE 1st
AND       M04161	// 16_R_2nd ROT T 2nd
AND       P00146	// R_2nd DIE VACUUM EJECTOR ON
OUT       M13040	// STEP A¢Ò¡ÆC17
MLOAD
AND       M13021	// 18.R_2nd ROT T 1st (Skip)
MPUSH
AND       M04140	// 14_R_2nd ROT Y IDLE 1st
AND       M04150	// 15_R_2nd ROT R IDLE 1st
AND       M04161	// 16_R_2nd ROT T 2nd
AND       P00146	// R_2nd DIE VACUUM EJECTOR ON
OUT       M13041	// STEP A¢Ò¡ÆC18
MPOP
AND       P00082	// R_2nd ALIGN CENTER FW
AND       P00083	// R_2nd ALIGN LEFT FW
AND NOT   P00084	// R_2nd SUPPORT UP FW
AND       P00085	// R_2nd PRESS RIGHT BW
AND NOT   P00086	// R_2nd PRESS RIGHT FW
AND       P00087	// R_2nd PRESS LEFT BW
AND NOT   P00088	// R_2nd PRESS LEFT FW
AND NOT   P00089	// R_2nd SUPPORT FW
AND       P0008A	// R_2nd SUPPORT BW
AND NOT   P0008B	// R_2nd SUPPORT SUB FW
AND       M04140	// 14_R_2nd ROT Y IDLE 1st
AND       M04150	// 15_R_2nd ROT R IDLE 1st
AND       M04160	// 16_R_2nd ROT T IDLE 1st
AND       P00146	// R_2nd DIE VACUUM EJECTOR ON
AND       F0009A
SET       P10000
MLOAD
AND       M13022	// 19.R_2nd ALIGN ALL BW
AND NOT   P00082	// R_2nd ALIGN CENTER FW
AND NOT   P00083	// R_2nd ALIGN LEFT FW
AND NOT   P00084	// R_2nd SUPPORT UP FW
AND       P00085	// R_2nd PRESS RIGHT BW
AND NOT   P00086	// R_2nd PRESS RIGHT FW
AND       P00087	// R_2nd PRESS LEFT BW
AND NOT   P00088	// R_2nd PRESS LEFT FW
AND NOT   P00089	// R_2nd SUPPORT FW
AND       P0008A	// R_2nd SUPPORT BW
AND NOT   P0008B	// R_2nd SUPPORT SUB FW
AND       M04140	// 14_R_2nd ROT Y IDLE 1st
AND       M04150	// 15_R_2nd ROT R IDLE 1st
AND       M04161	// 16_R_2nd ROT T 2nd
AND       P00146	// R_2nd DIE VACUUM EJECTOR ON
OUT       M13042	// STEP A¢Ò¡ÆC19
MLOAD
AND       M13023	// -
OUT       M13043	// STEP A¢Ò¡ÆC20
MLOAD
AND       M13024	// -
OUT       M13044	// STEP A¢Ò¡ÆC21
MLOAD
AND       M13025	// -
OUT       M13045	// STEP A¢Ò¡ÆC22
MLOAD
AND       M13026	// -
OUT       M13046	// STEP A¢Ò¡ÆC23
MLOAD
AND       M13027	// -
OUT       M13047	// STEP A¢Ò¡ÆC24
MLOAD
AND       M13028	// -
OUT       M13048	// STEP A¢Ò¡ÆC25
MLOAD
AND       M13029	// -
OUT       M13049	// STEP A¢Ò¡ÆC26
MLOAD
AND       M1302A	// -
OUT       M1304A	// STEP A¢Ò¡ÆC27
MLOAD
AND       M1302B	// -
OUT       M1304B	// STEP A¢Ò¡ÆC28
MLOAD
AND       M1302C	// -
OUT       M1304C	// STEP A¢Ò¡ÆC29
MLOAD
AND       M1302D	// -
OUT       M1304D	// STEP A¢Ò¡ÆC30
MLOAD
AND       M1302E	// -
OUT       M1304E	// STEP A¢Ò¡ÆC31
MPOP
AND       M1302F	// 32.R_2nd STEP END
OUT       M1304F	// STEP A¢Ò¡ÆC32
DMOV      2147483648 M1301

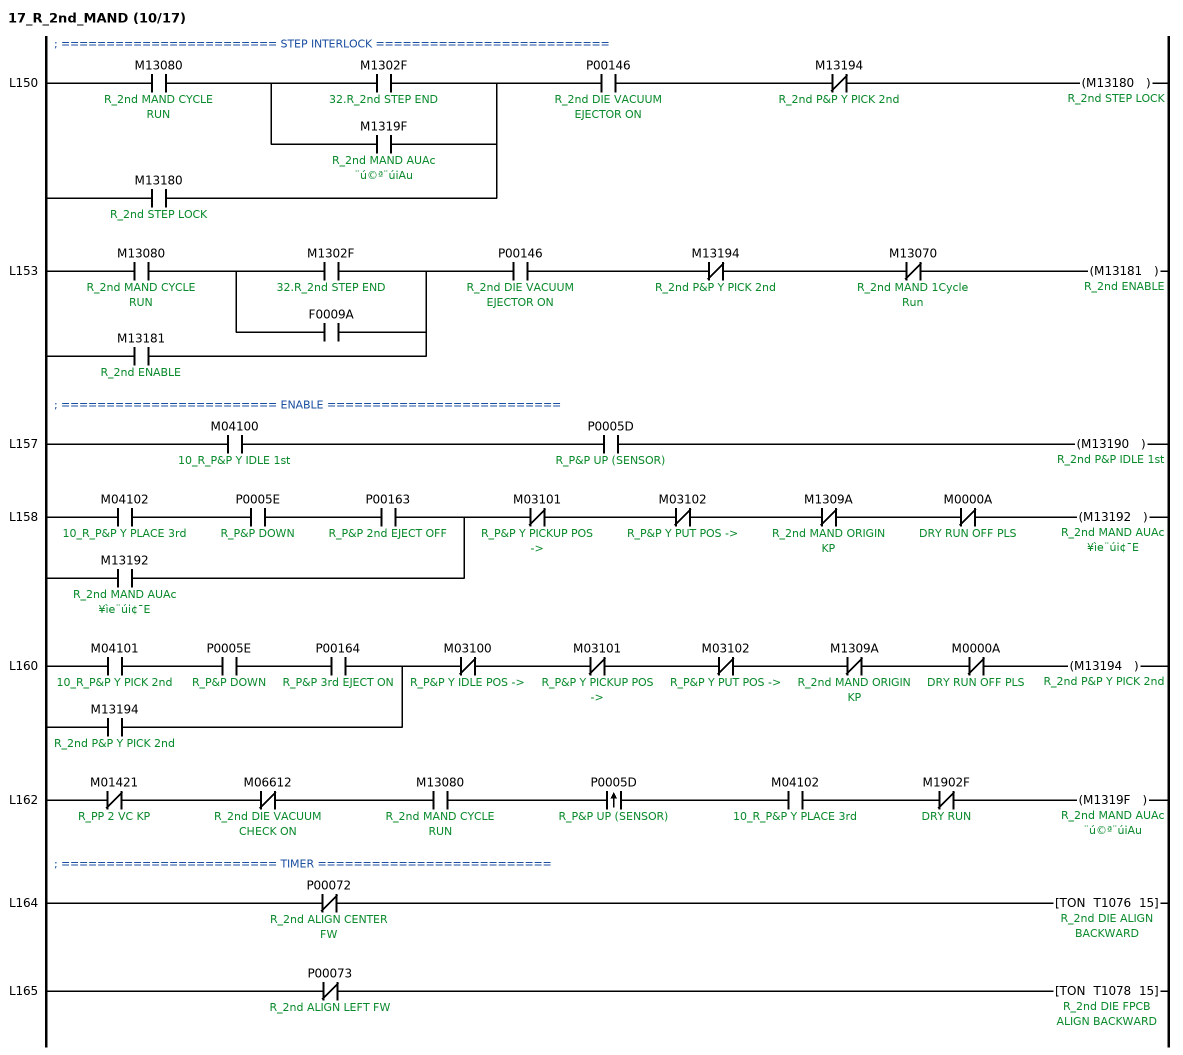
// ======================== STEP INTERLOCK ==========================
; L150
LOAD      M13080	// R_2nd MAND CYCLE RUN
LOAD      M1302F	// 32.R_2nd STEP END
OR        M1319F	// R_2nd MAND AUAc ¨ú©ª¨úiAu
AND LOAD
OR        M13180	// R_2nd STEP LOCK
AND       P00146	// R_2nd DIE VACUUM EJECTOR ON
AND NOT   M13194	// R_2nd P&P Y PICK 2nd
OUT       M13180	// R_2nd STEP LOCK
; L153
LOAD      M13080	// R_2nd MAND CYCLE RUN
LOAD      M1302F	// 32.R_2nd STEP END
OR        F0009A
AND LOAD
OR        M13181	// R_2nd ENABLE
AND       P00146	// R_2nd DIE VACUUM EJECTOR ON
AND NOT   M13194	// R_2nd P&P Y PICK 2nd
AND NOT   M13070	// R_2nd MAND 1Cycle Run
OUT       M13181	// R_2nd ENABLE
// ======================== ENABLE ==========================
; L157
LOAD      M04100	// 10_R_P&P Y IDLE 1st
AND       P0005D	// R_P&P UP (SENSOR)
OUT       M13190	// R_2nd P&P IDLE 1st
; L158
LOAD      M04102	// 10_R_P&P Y PLACE 3rd
AND       P0005E	// R_P&P DOWN
AND       P00163	// R_P&P 2nd EJECT OFF
OR        M13192	// R_2nd MAND AUAc ¥ìe¨úi¢¯E
AND NOT   M03101	// R_P&P Y PICKUP POS ->
AND NOT   M03102	// R_P&P Y PUT POS ->
AND NOT   M1309A	// R_2nd MAND ORIGIN KP
AND NOT   M0000A	// DRY RUN OFF PLS
OUT       M13192	// R_2nd MAND AUAc ¥ìe¨úi¢¯E
; L160
LOAD      M04101	// 10_R_P&P Y PICK 2nd
AND       P0005E	// R_P&P DOWN
AND       P00164	// R_P&P 3rd EJECT ON
OR        M13194	// R_2nd P&P Y PICK 2nd
AND NOT   M03100	// R_P&P Y IDLE POS ->
AND NOT   M03101	// R_P&P Y PICKUP POS ->
AND NOT   M03102	// R_P&P Y PUT POS ->
AND NOT   M1309A	// R_2nd MAND ORIGIN KP
AND NOT   M0000A	// DRY RUN OFF PLS
OUT       M13194	// R_2nd P&P Y PICK 2nd
; L162
LOAD NOT  M01421	// R_PP 2 VC KP
AND NOT   M06612	// R_2nd DIE VACUUM CHECK ON
AND       M13080	// R_2nd MAND CYCLE RUN
ANDP      P0005D	// R_P&P UP (SENSOR)
AND       M04102	// 10_R_P&P Y PLACE 3rd
AND NOT   M1902F	// DRY RUN
OUT       M1319F	// R_2nd MAND AUAc ¨ú©ª¨úiAu
// ======================== TIMER ==========================
; L164
LOAD NOT  P00072	// R_2nd ALIGN CENTER FW
TON       T1076 15	// R_2nd DIE ALIGN BACKWARD
; L165
LOAD NOT  P00073	// R_2nd ALIGN LEFT FW
TON       T1078 15	// R_2nd DIE FPCB ALIGN BACKWARD

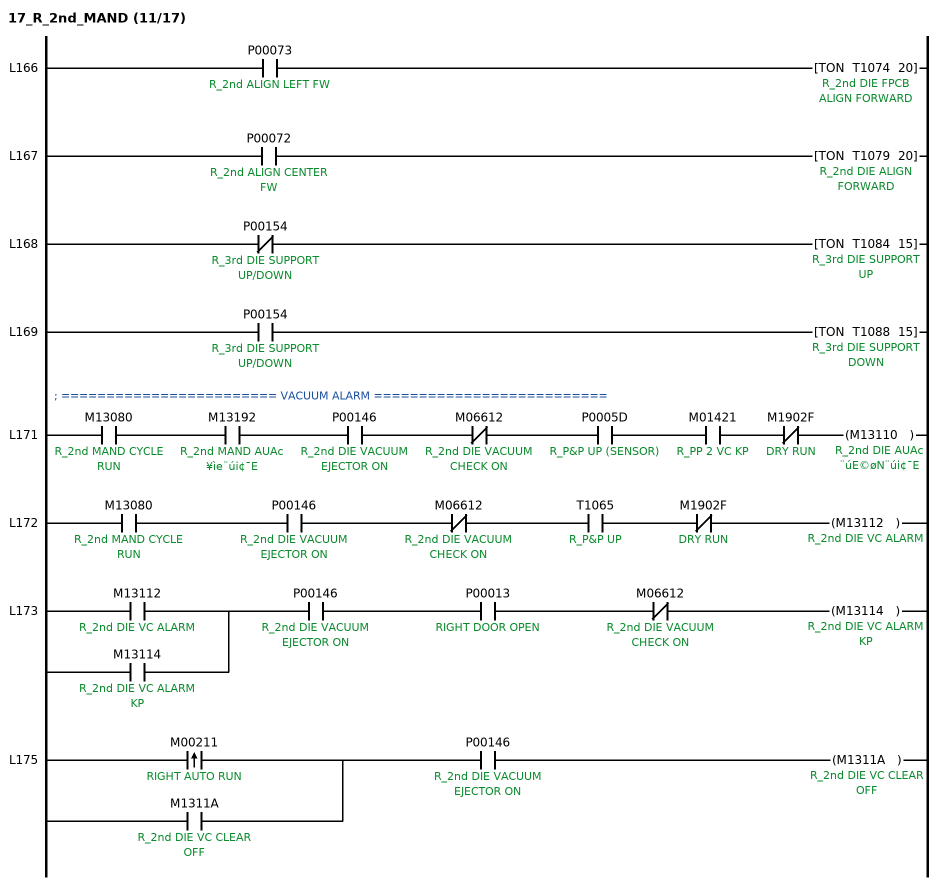
; L166
LOAD      P00073	// R_2nd ALIGN LEFT FW
TON       T1074 20	// R_2nd DIE FPCB ALIGN FORWARD
; L167
LOAD      P00072	// R_2nd ALIGN CENTER FW
TON       T1079 20	// R_2nd DIE ALIGN FORWARD
; L168
LOAD NOT  P00154	// R_3rd DIE SUPPORT UP/DOWN
TON       T1084 15	// R_3rd DIE SUPPORT UP
; L169
LOAD      P00154	// R_3rd DIE SUPPORT UP/DOWN
TON       T1088 15	// R_3rd DIE SUPPORT DOWN
// ======================== VACUUM ALARM ==========================
; L171
LOAD      M13080	// R_2nd MAND CYCLE RUN
AND       M13192	// R_2nd MAND AUAc ¥ìe¨úi¢¯E
AND       P00146	// R_2nd DIE VACUUM EJECTOR ON
AND NOT   M06612	// R_2nd DIE VACUUM CHECK ON
AND       P0005D	// R_P&P UP (SENSOR)
AND       M01421	// R_PP 2 VC KP
AND NOT   M1902F	// DRY RUN
OUT       M13110	// R_2nd DIE AUAc ¨úE©øN¨úi¢¯E
; L172
LOAD      M13080	// R_2nd MAND CYCLE RUN
AND       P00146	// R_2nd DIE VACUUM EJECTOR ON
AND NOT   M06612	// R_2nd DIE VACUUM CHECK ON
AND       T1065	// R_P&P UP
AND NOT   M1902F	// DRY RUN
OUT       M13112	// R_2nd DIE VC ALARM
; L173
LOAD      M13112	// R_2nd DIE VC ALARM
OR        M13114	// R_2nd DIE VC ALARM KP
AND       P00146	// R_2nd DIE VACUUM EJECTOR ON
AND       P00013	// RIGHT DOOR OPEN
AND NOT   M06612	// R_2nd DIE VACUUM CHECK ON
OUT       M13114	// R_2nd DIE VC ALARM KP
; L175
LOADP     M00211	// RIGHT AUTO RUN
OR        M1311A	// R_2nd DIE VC CLEAR OFF
AND       P00146	// R_2nd DIE VACUUM EJECTOR ON
OUT       M1311A	// R_2nd DIE VC CLEAR OFF

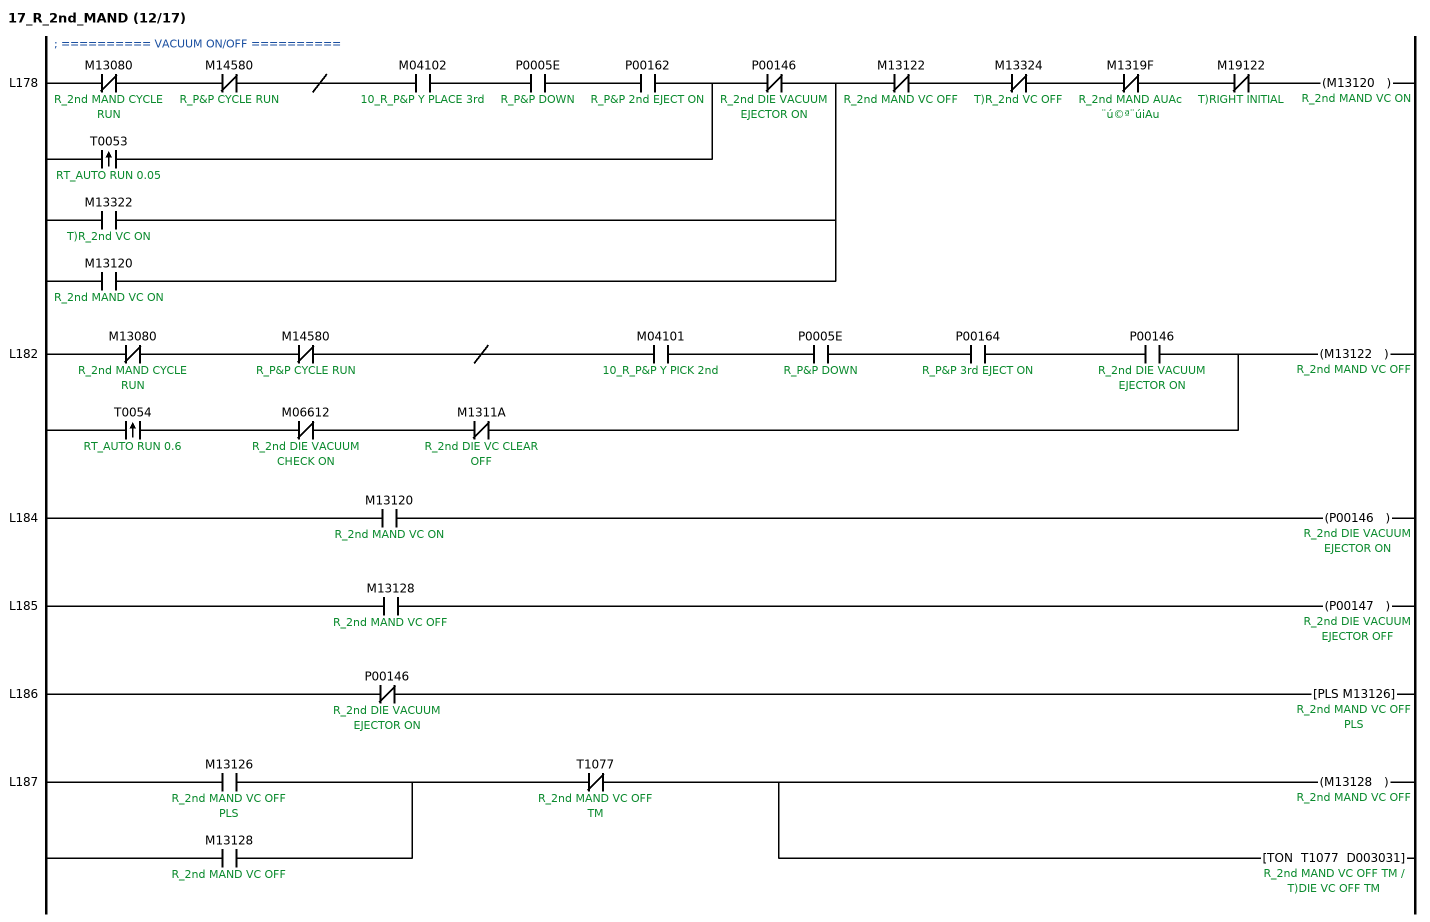
// ========== VACUUM ON/OFF ==========
; L178
LOAD NOT  M13080	// R_2nd MAND CYCLE RUN
AND NOT   M14580	// R_P&P CYCLE RUN
NOT
AND       M04102	// 10_R_P&P Y PLACE 3rd
AND       P0005E	// R_P&P DOWN
AND       P00162	// R_P&P 2nd EJECT ON
ORP       T0053	// RT_AUTO RUN 0.05
AND NOT   P00146	// R_2nd DIE VACUUM EJECTOR ON
OR        M13322	// T)R_2nd VC ON
OR        M13120	// R_2nd MAND VC ON
AND NOT   M13122	// R_2nd MAND VC OFF
AND NOT   M13324	// T)R_2nd VC OFF
AND NOT   M1319F	// R_2nd MAND AUAc ¨ú©ª¨úiAu
AND NOT   M19122	// T)RIGHT INITIAL
OUT       M13120	// R_2nd MAND VC ON
; L182
LOAD NOT  M13080	// R_2nd MAND CYCLE RUN
AND NOT   M14580	// R_P&P CYCLE RUN
NOT
AND       M04101	// 10_R_P&P Y PICK 2nd
AND       P0005E	// R_P&P DOWN
AND       P00164	// R_P&P 3rd EJECT ON
AND       P00146	// R_2nd DIE VACUUM EJECTOR ON
LOADP     T0054	// RT_AUTO RUN 0.6
AND NOT   M06612	// R_2nd DIE VACUUM CHECK ON
AND NOT   M1311A	// R_2nd DIE VC CLEAR OFF
OR LOAD
OUT       M13122	// R_2nd MAND VC OFF
; L184
LOAD      M13120	// R_2nd MAND VC ON
OUT       P00146	// R_2nd DIE VACUUM EJECTOR ON
; L185
LOAD      M13128	// R_2nd MAND VC OFF
OUT       P00147	// R_2nd DIE VACUUM EJECTOR OFF
; L186
LOAD NOT  P00146	// R_2nd DIE VACUUM EJECTOR ON
OUTP      M13126	// R_2nd MAND VC OFF PLS
; L187
LOAD      M13126	// R_2nd MAND VC OFF PLS
OR        M13128	// R_2nd MAND VC OFF
AND NOT   T1077	// R_2nd MAND VC OFF TM
OUT       M13128	// R_2nd MAND VC OFF
TON       T1077 D003031	// R_2nd MAND VC OFF TM / T)DIE VC OFF TM

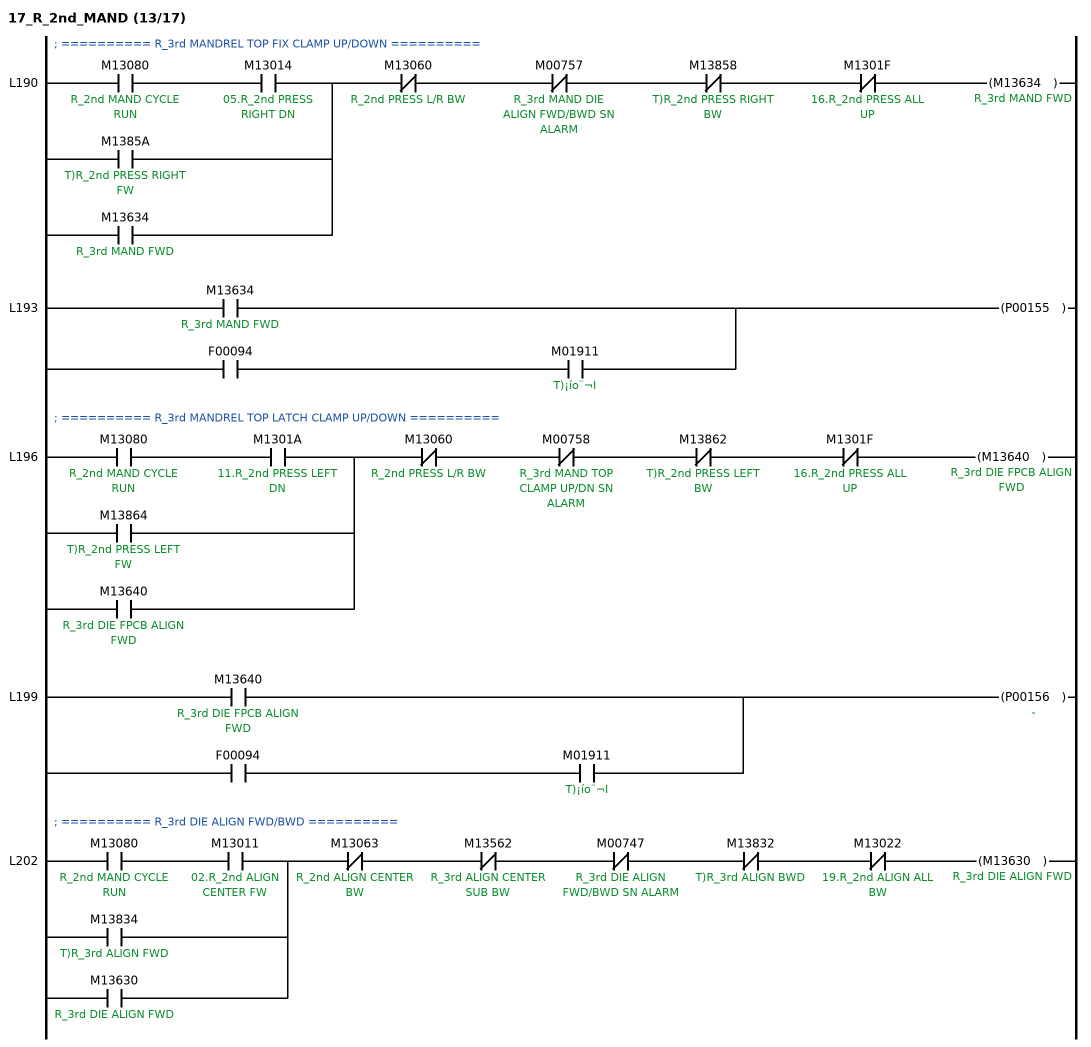
// ========== R_3rd MANDREL TOP FIX CLAMP UP/DOWN ==========
; L190
LOAD      M13080	// R_2nd MAND CYCLE RUN
AND       M13014	// 05.R_2nd PRESS RIGHT DN
OR        M1385A	// T)R_2nd PRESS RIGHT FW
OR        M13634	// R_3rd MAND FWD
AND NOT   M13060	// R_2nd PRESS L/R BW
AND NOT   M00757	// R_3rd MAND DIE ALIGN FWD/BWD SN ALARM
AND NOT   M13858	// T)R_2nd PRESS RIGHT BW
AND NOT   M1301F	// 16.R_2nd PRESS ALL UP
OUT       M13634	// R_3rd MAND FWD
; L193
LOAD      M13634	// R_3rd MAND FWD
LOAD      F00094
AND       M01911	// T)¡ío¨¬I
OR LOAD
OUT       P00155
// ========== R_3rd MANDREL TOP LATCH CLAMP UP/DOWN ==========
; L196
LOAD      M13080	// R_2nd MAND CYCLE RUN
AND       M1301A	// 11.R_2nd PRESS LEFT DN
OR        M13864	// T)R_2nd PRESS LEFT FW
OR        M13640	// R_3rd DIE FPCB ALIGN FWD
AND NOT   M13060	// R_2nd PRESS L/R BW
AND NOT   M00758	// R_3rd MAND TOP CLAMP UP/DN SN ALARM
AND NOT   M13862	// T)R_2nd PRESS LEFT BW
AND NOT   M1301F	// 16.R_2nd PRESS ALL UP
OUT       M13640	// R_3rd DIE FPCB ALIGN FWD
; L199
LOAD      M13640	// R_3rd DIE FPCB ALIGN FWD
LOAD      F00094
AND       M01911	// T)¡ío¨¬I
OR LOAD
OUT       P00156	// -
// ========== R_3rd DIE ALIGN FWD/BWD ==========
; L202
LOAD      M13080	// R_2nd MAND CYCLE RUN
AND       M13011	// 02.R_2nd ALIGN CENTER FW
OR        M13834	// T)R_3rd ALIGN FWD
OR        M13630	// R_3rd DIE ALIGN FWD
AND NOT   M13063	// R_2nd ALIGN CENTER BW
AND NOT   M13562	// R_3rd ALIGN CENTER SUB BW
AND NOT   M00747	// R_3rd DIE ALIGN FWD/BWD SN ALARM
AND NOT   M13832	// T)R_3rd ALIGN BWD
AND NOT   M13022	// 19.R_2nd ALIGN ALL BW
OUT       M13630	// R_3rd DIE ALIGN FWD

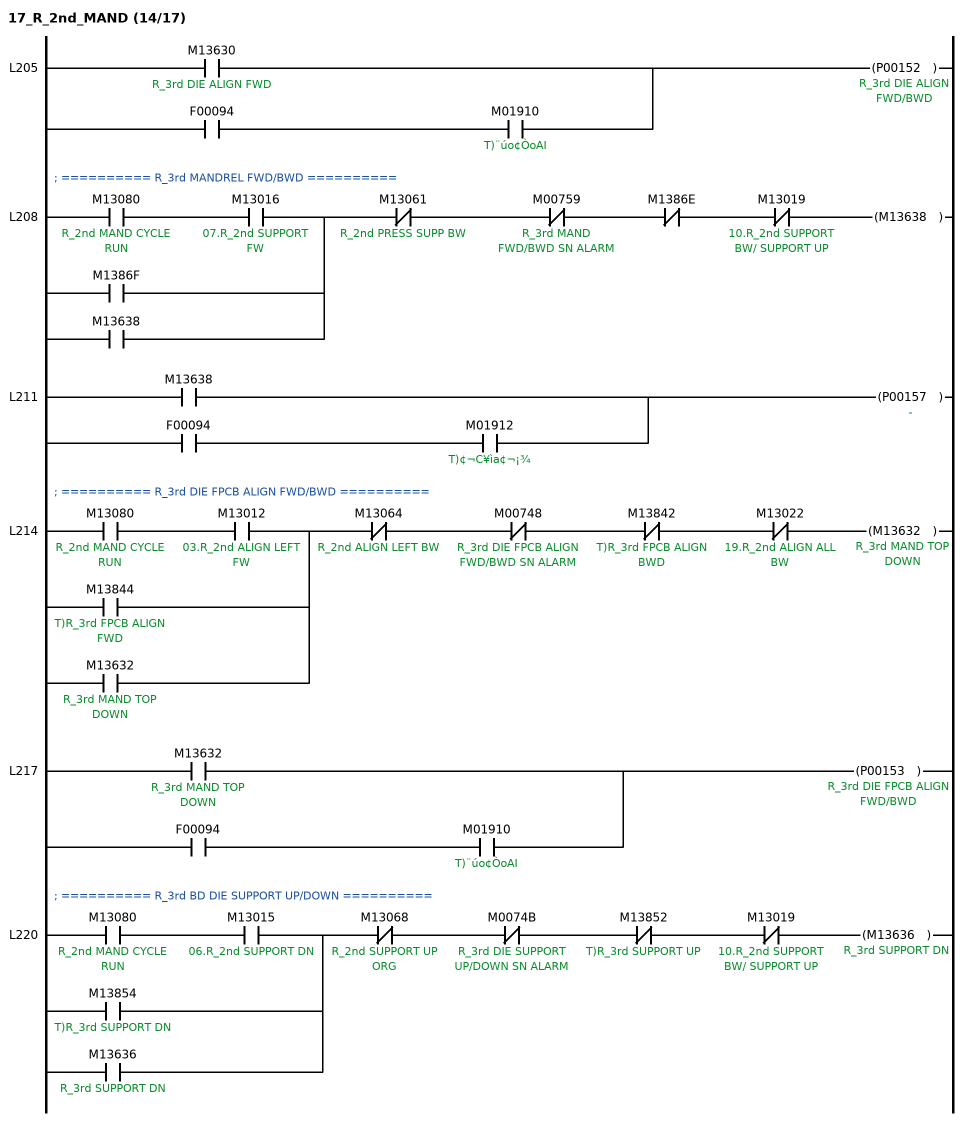
; L205
LOAD      M13630	// R_3rd DIE ALIGN FWD
LOAD      F00094
AND       M01910	// T)¨úo¢ÒoAI
OR LOAD
OUT       P00152	// R_3rd DIE ALIGN FWD/BWD
// ========== R_3rd MANDREL FWD/BWD ==========
; L208
LOAD      M13080	// R_2nd MAND CYCLE RUN
AND       M13016	// 07.R_2nd SUPPORT FW
OR        M1386F
OR        M13638
AND NOT   M13061	// R_2nd PRESS SUPP BW
AND NOT   M00759	// R_3rd MAND FWD/BWD SN ALARM
AND NOT   M1386E
AND NOT   M13019	// 10.R_2nd SUPPORT BW/ SUPPORT UP
OUT       M13638
; L211
LOAD      M13638
LOAD      F00094
AND       M01912	// T)¢¬C¥ìa¢¬¡¾
OR LOAD
OUT       P00157	// -
// ========== R_3rd DIE FPCB ALIGN FWD/BWD ==========
; L214
LOAD      M13080	// R_2nd MAND CYCLE RUN
AND       M13012	// 03.R_2nd ALIGN LEFT FW
OR        M13844	// T)R_3rd FPCB ALIGN FWD
OR        M13632	// R_3rd MAND TOP DOWN
AND NOT   M13064	// R_2nd ALIGN LEFT BW
AND NOT   M00748	// R_3rd DIE FPCB ALIGN FWD/BWD SN ALARM
AND NOT   M13842	// T)R_3rd FPCB ALIGN BWD
AND NOT   M13022	// 19.R_2nd ALIGN ALL BW
OUT       M13632	// R_3rd MAND TOP DOWN
; L217
LOAD      M13632	// R_3rd MAND TOP DOWN
LOAD      F00094
AND       M01910	// T)¨úo¢ÒoAI
OR LOAD
OUT       P00153	// R_3rd DIE FPCB ALIGN FWD/BWD
// ========== R_3rd BD DIE SUPPORT UP/DOWN ==========
; L220
LOAD      M13080	// R_2nd MAND CYCLE RUN
AND       M13015	// 06.R_2nd SUPPORT DN
OR        M13854	// T)R_3rd SUPPORT DN
OR        M13636	// R_3rd SUPPORT DN
AND NOT   M13068	// R_2nd SUPPORT UP ORG
AND NOT   M0074B	// R_3rd DIE SUPPORT UP/DOWN SN ALARM
AND NOT   M13852	// T)R_3rd SUPPORT UP
AND NOT   M13019	// 10.R_2nd SUPPORT BW/ SUPPORT UP
OUT       M13636	// R_3rd SUPPORT DN

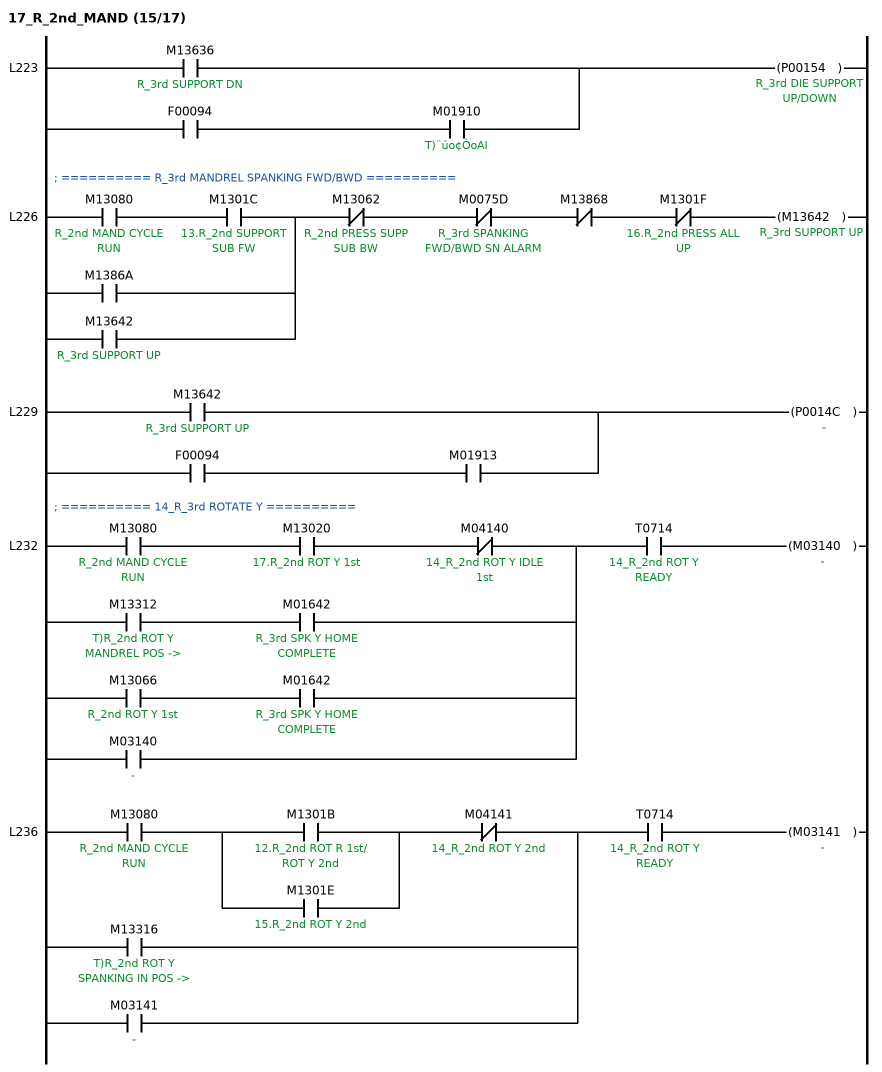
; L223
LOAD      M13636	// R_3rd SUPPORT DN
LOAD      F00094
AND       M01910	// T)¨úo¢ÒoAI
OR LOAD
OUT       P00154	// R_3rd DIE SUPPORT UP/DOWN
// ========== R_3rd MANDREL SPANKING FWD/BWD ==========
; L226
LOAD      M13080	// R_2nd MAND CYCLE RUN
AND       M1301C	// 13.R_2nd SUPPORT SUB FW
OR        M1386A
OR        M13642	// R_3rd SUPPORT UP
AND NOT   M13062	// R_2nd PRESS SUPP SUB BW
AND NOT   M0075D	// R_3rd SPANKING FWD/BWD SN ALARM
AND NOT   M13868
AND NOT   M1301F	// 16.R_2nd PRESS ALL UP
OUT       M13642	// R_3rd SUPPORT UP
; L229
LOAD      M13642	// R_3rd SUPPORT UP
LOAD      F00094
AND       M01913
OR LOAD
OUT       P0014C	// -
// ========== 14_R_3rd ROTATE Y ==========
; L232
LOAD      M13080	// R_2nd MAND CYCLE RUN
AND       M13020	// 17.R_2nd ROT Y 1st
AND NOT   M04140	// 14_R_2nd ROT Y IDLE 1st
LOAD      M13312	// T)R_2nd ROT Y MANDREL POS ->
AND       M01642	// R_3rd SPK Y HOME COMPLETE
OR LOAD
LOAD      M13066	// R_2nd ROT Y 1st
AND       M01642	// R_3rd SPK Y HOME COMPLETE
OR LOAD
OR        M03140	// -
AND       T0714	// 14_R_2nd ROT Y READY
OUT       M03140	// -
; L236
LOAD      M13080	// R_2nd MAND CYCLE RUN
LOAD      M1301B	// 12.R_2nd ROT R 1st/ ROT Y 2nd
OR        M1301E	// 15.R_2nd ROT Y 2nd
AND LOAD
AND NOT   M04141	// 14_R_2nd ROT Y 2nd
OR        M13316	// T)R_2nd ROT Y SPANKING IN POS ->
OR        M03141	// -
AND       T0714	// 14_R_2nd ROT Y READY
OUT       M03141	// -

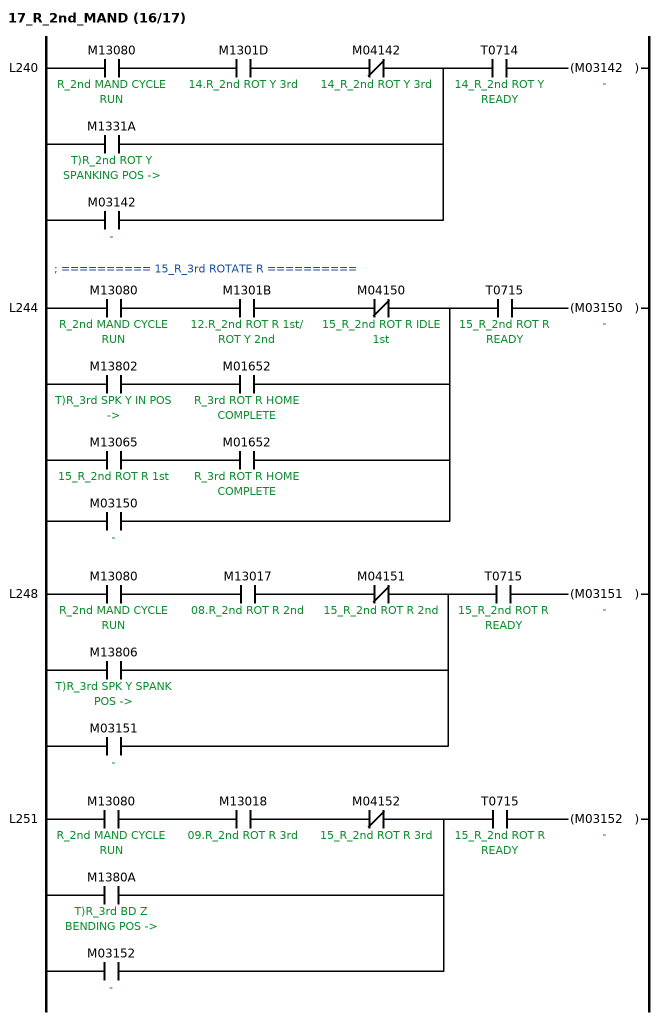
; L240
LOAD      M13080	// R_2nd MAND CYCLE RUN
AND       M1301D	// 14.R_2nd ROT Y 3rd
AND NOT   M04142	// 14_R_2nd ROT Y 3rd
OR        M1331A	// T)R_2nd ROT Y SPANKING POS ->
OR        M03142	// -
AND       T0714	// 14_R_2nd ROT Y READY
OUT       M03142	// -
// ========== 15_R_3rd ROTATE R ==========
; L244
LOAD      M13080	// R_2nd MAND CYCLE RUN
AND       M1301B	// 12.R_2nd ROT R 1st/ ROT Y 2nd
AND NOT   M04150	// 15_R_2nd ROT R IDLE 1st
LOAD      M13802	// T)R_3rd SPK Y IN POS ->
AND       M01652	// R_3rd ROT R HOME COMPLETE
OR LOAD
LOAD      M13065	// 15_R_2nd ROT R 1st
AND       M01652	// R_3rd ROT R HOME COMPLETE
OR LOAD
OR        M03150	// -
AND       T0715	// 15_R_2nd ROT R READY
OUT       M03150	// -
; L248
LOAD      M13080	// R_2nd MAND CYCLE RUN
AND       M13017	// 08.R_2nd ROT R 2nd
AND NOT   M04151	// 15_R_2nd ROT R 2nd
OR        M13806	// T)R_3rd SPK Y SPANK POS ->
OR        M03151	// -
AND       T0715	// 15_R_2nd ROT R READY
OUT       M03151	// -
; L251
LOAD      M13080	// R_2nd MAND CYCLE RUN
AND       M13018	// 09.R_2nd ROT R 3rd
AND NOT   M04152	// 15_R_2nd ROT R 3rd
OR        M1380A	// T)R_3rd BD Z BENDING POS ->
OR        M03152	// -
AND       T0715	// 15_R_2nd ROT R READY
OUT       M03152	// -

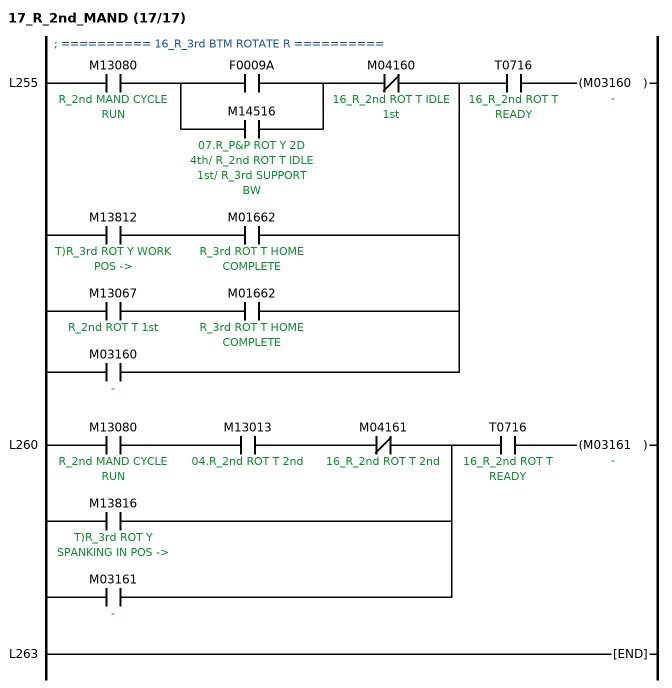
// ========== 16_R_3rd BTM ROTATE R ==========
; L255
LOAD      M13080	// R_2nd MAND CYCLE RUN
LOAD      F0009A
OR        M14516	// 07.R_P&P ROT Y 2D 4th/ R_2nd ROT T IDLE 1st/ R_3rd SUPPORT BW
AND LOAD
AND NOT   M04160	// 16_R_2nd ROT T IDLE 1st
LOAD      M13812	// T)R_3rd ROT Y WORK POS ->
AND       M01662	// R_3rd ROT T HOME COMPLETE
OR LOAD
LOAD      M13067	// R_2nd ROT T 1st
AND       M01662	// R_3rd ROT T HOME COMPLETE
OR LOAD
OR        M03160	// -
AND       T0716	// 16_R_2nd ROT T READY
OUT       M03160	// -
; L260
LOAD      M13080	// R_2nd MAND CYCLE RUN
AND       M13013	// 04.R_2nd ROT T 2nd
AND NOT   M04161	// 16_R_2nd ROT T 2nd
OR        M13816	// T)R_3rd ROT Y SPANKING IN POS ->
OR        M03161	// -
AND       T0716	// 16_R_2nd ROT T READY
OUT       M03161	// -
; L263
END

PROGRAM 18_R_3rd_MAND (task: ¨ö¨¬A¥ì CA¡¤I¡¾¡¿¡¤¡Í)

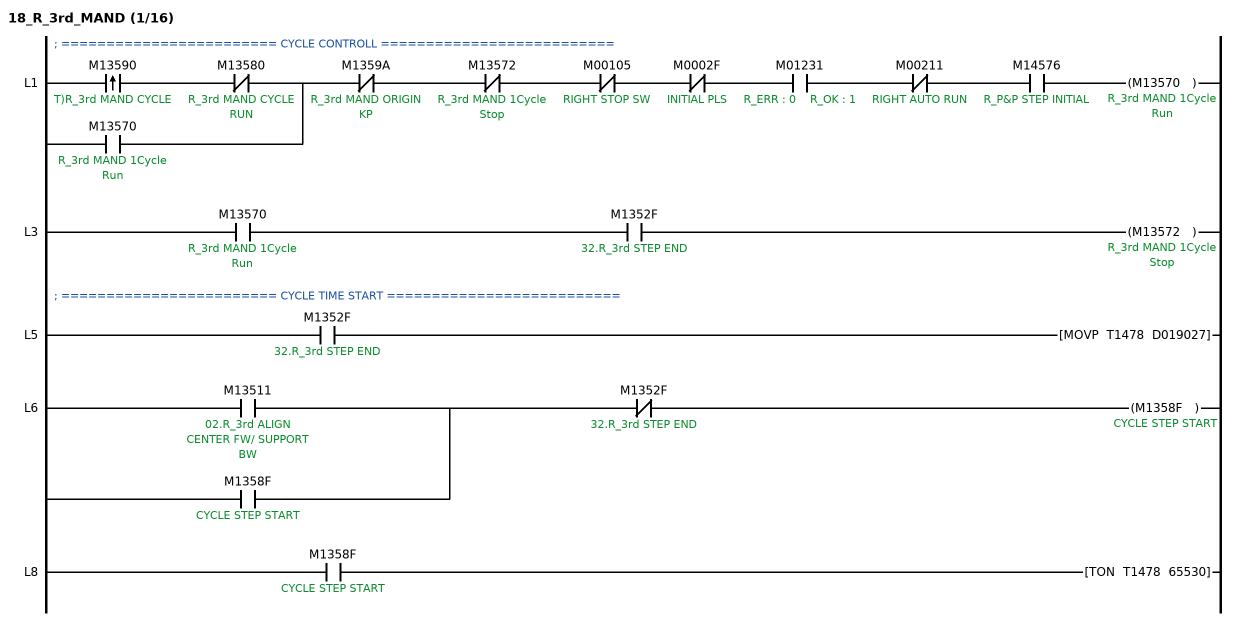
// ======================== CYCLE CONTROLL ==========================
; L1
LOADP     M13590	// T)R_3rd MAND CYCLE
AND NOT   M13580	// R_3rd MAND CYCLE RUN
OR        M13570	// R_3rd MAND 1Cycle Run
AND NOT   M1359A	// R_3rd MAND ORIGIN KP
AND NOT   M13572	// R_3rd MAND 1Cycle Stop
AND NOT   M00105	// RIGHT STOP SW
AND NOT   M0002F	// INITIAL PLS
AND       M01231	// R_ERR : 0    R_OK : 1
AND NOT   M00211	// RIGHT AUTO RUN
AND       M14576	// R_P&P STEP INITIAL
OUT       M13570	// R_3rd MAND 1Cycle Run
; L3
LOAD      M13570	// R_3rd MAND 1Cycle Run
AND       M1352F	// 32.R_3rd STEP END
OUT       M13572	// R_3rd MAND 1Cycle Stop
// ======================== CYCLE TIME START ==========================
; L5
LOAD      M1352F	// 32.R_3rd STEP END
MOVP      T1478 D019027
; L6
LOAD      M13511	// 02.R_3rd ALIGN CENTER FW/ SUPPORT BW
OR        M1358F	// CYCLE STEP START
AND NOT   M1352F	// 32.R_3rd STEP END
OUT       M1358F	// CYCLE STEP START
; L8
LOAD      M1358F	// CYCLE STEP START
TON       T1478 65530

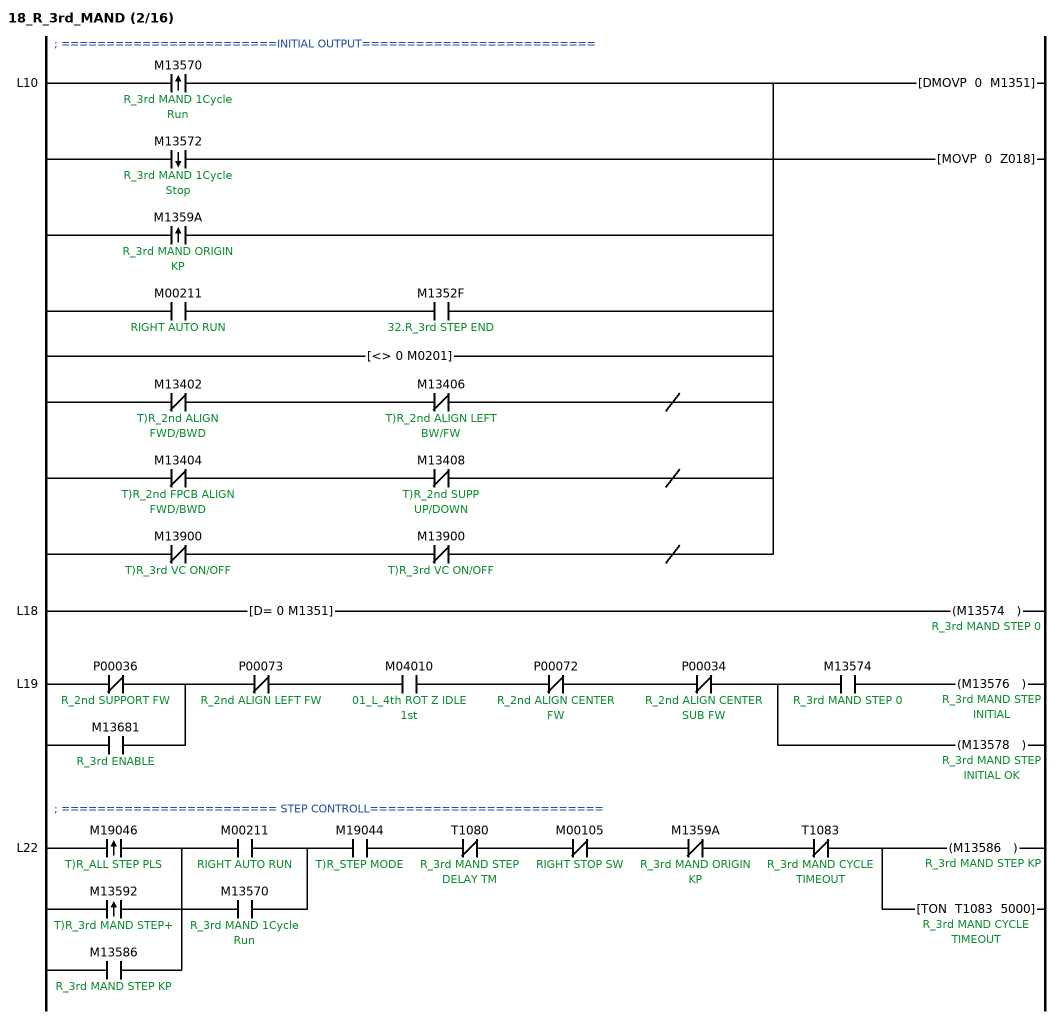
// ========================INITIAL OUTPUT==========================
; L10
LOADP     M13570	// R_3rd MAND 1Cycle Run
ORN       M13572	// R_3rd MAND 1Cycle Stop
ORP       M1359A	// R_3rd MAND ORIGIN KP
LOAD      M00211	// RIGHT AUTO RUN
AND       M1352F	// 32.R_3rd STEP END
OR LOAD
OR<>      0 M0201
LOAD NOT  M13402	// T)R_2nd ALIGN FWD/BWD
AND NOT   M13406	// T)R_2nd ALIGN LEFT BW/FW
NOT
OR LOAD
LOAD NOT  M13404	// T)R_2nd FPCB ALIGN FWD/BWD
AND NOT   M13408	// T)R_2nd SUPP UP/DOWN
NOT
OR LOAD
LOAD NOT  M13900	// T)R_3rd VC ON/OFF
AND NOT   M13900	// T)R_3rd VC ON/OFF
NOT
OR LOAD
DMOVP     0 M1351
MOVP      0 Z018
; L18
LOADD=    0 M1351
OUT       M13574	// R_3rd MAND STEP 0
; L19
LOAD NOT  P00036	// R_2nd SUPPORT FW
OR        M13681	// R_3rd ENABLE
AND NOT   P00073	// R_2nd ALIGN LEFT FW
AND       M04010	// 01_L_4th ROT Z IDLE 1st
AND NOT   P00072	// R_2nd ALIGN CENTER FW
AND NOT   P00034	// R_2nd ALIGN CENTER SUB FW
MPUSH
AND       M13574	// R_3rd MAND STEP 0
OUT       M13576	// R_3rd MAND STEP INITIAL
MPOP
OUT       M13578	// R_3rd MAND STEP INITIAL OK
// ======================== STEP CONTROLL==========================
; L22
LOADP     M19046	// T)R_ALL STEP PLS
ORP       M13592	// T)R_3rd MAND STEP+
OR        M13586	// R_3rd MAND STEP KP
LOAD      M00211	// RIGHT AUTO RUN
OR        M13570	// R_3rd MAND 1Cycle Run
AND LOAD
AND       M19044	// T)R_STEP MODE
AND NOT   T1080	// R_3rd MAND STEP DELAY TM
AND NOT   M00105	// RIGHT STOP SW
AND NOT   M1359A	// R_3rd MAND ORIGIN KP
AND NOT   T1083	// R_3rd MAND CYCLE TIMEOUT
OUT       M13586	// R_3rd MAND STEP KP
TON       T1083 5000	// R_3rd MAND CYCLE TIMEOUT

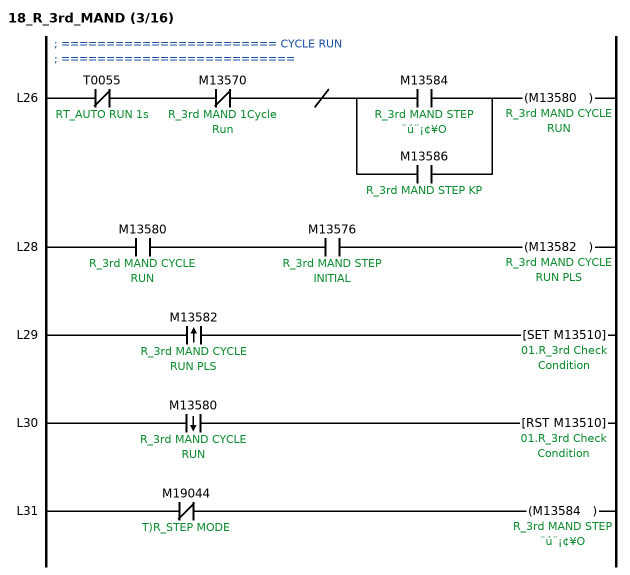
// ======================== CYCLE RUN ==========================
; L26
LOAD NOT  T0055	// RT_AUTO RUN 1s
AND NOT   M13570	// R_3rd MAND 1Cycle Run
NOT
LOAD      M13584	// R_3rd MAND STEP ¨ú¨¡¢¥O
OR        M13586	// R_3rd MAND STEP KP
AND LOAD
OUT       M13580	// R_3rd MAND CYCLE RUN
; L28
LOAD      M13580	// R_3rd MAND CYCLE RUN
AND       M13576	// R_3rd MAND STEP INITIAL
OUT       M13582	// R_3rd MAND CYCLE RUN PLS
; L29
LOADP     M13582	// R_3rd MAND CYCLE RUN PLS
SET       M13510	// 01.R_3rd Check Condition
; L30
LOADN     M13580	// R_3rd MAND CYCLE RUN
RST       M13510	// 01.R_3rd Check Condition
; L31
LOAD NOT  M19044	// T)R_STEP MODE
OUT       M13584	// R_3rd MAND STEP ¨ú¨¡¢¥O

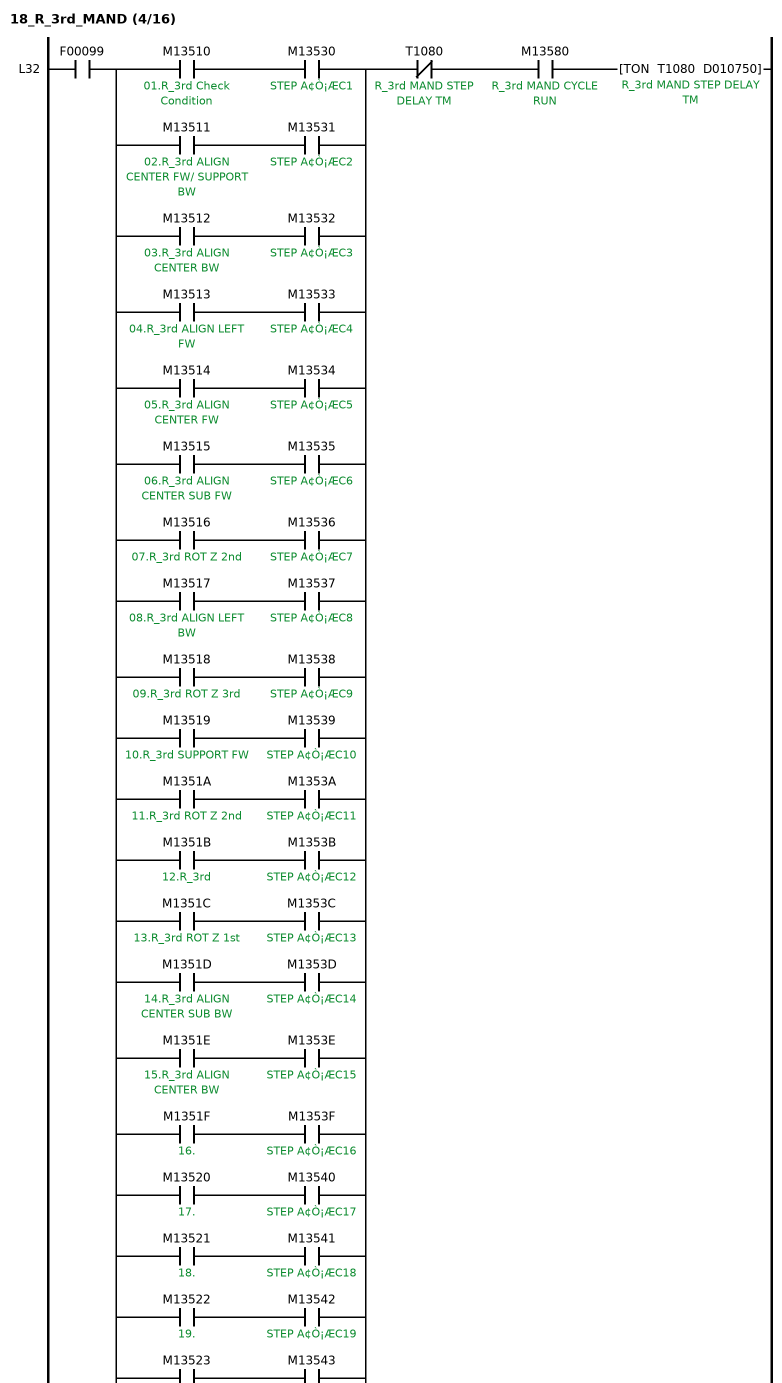

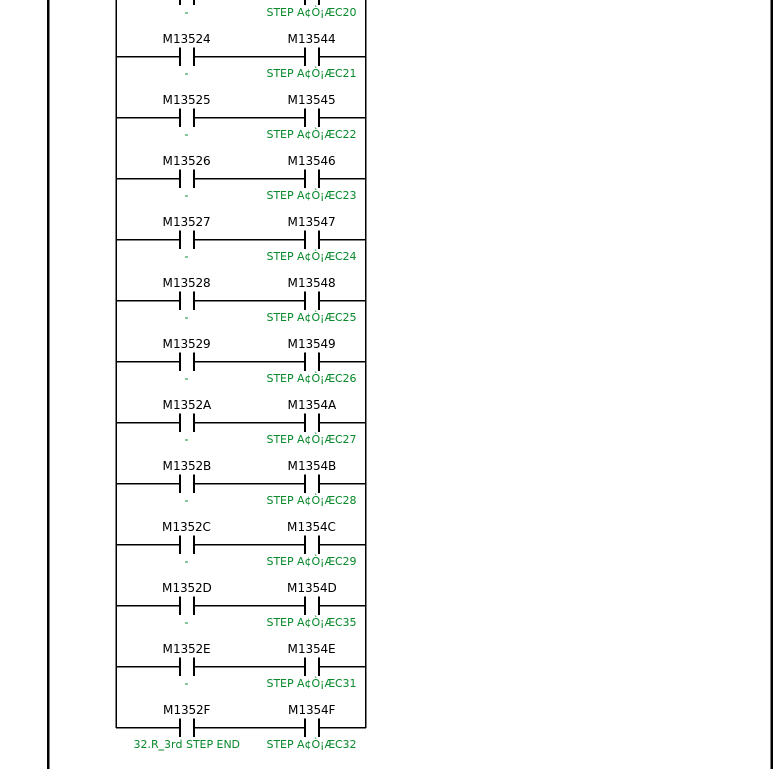
; L32
LOAD      F00099
LOAD      M13510	// 01.R_3rd Check Condition
AND       M13530	// STEP A¢Ò¡ÆC1
LOAD      M13511	// 02.R_3rd ALIGN CENTER FW/ SUPPORT BW
AND       M13531	// STEP A¢Ò¡ÆC2
OR LOAD
LOAD      M13512	// 03.R_3rd ALIGN CENTER BW
AND       M13532	// STEP A¢Ò¡ÆC3
OR LOAD
LOAD      M13513	// 04.R_3rd ALIGN LEFT FW
AND       M13533	// STEP A¢Ò¡ÆC4
OR LOAD
LOAD      M13514	// 05.R_3rd ALIGN CENTER FW
AND       M13534	// STEP A¢Ò¡ÆC5
OR LOAD
LOAD      M13515	// 06.R_3rd ALIGN CENTER SUB FW
AND       M13535	// STEP A¢Ò¡ÆC6
OR LOAD
LOAD      M13516	// 07.R_3rd ROT Z 2nd
AND       M13536	// STEP A¢Ò¡ÆC7
OR LOAD
LOAD      M13517	// 08.R_3rd ALIGN LEFT BW
AND       M13537	// STEP A¢Ò¡ÆC8
OR LOAD
LOAD      M13518	// 09.R_3rd ROT Z 3rd
AND       M13538	// STEP A¢Ò¡ÆC9
OR LOAD
LOAD      M13519	// 10.R_3rd SUPPORT FW
AND       M13539	// STEP A¢Ò¡ÆC10
OR LOAD
LOAD      M1351A	// 11.R_3rd ROT Z 2nd
AND       M1353A	// STEP A¢Ò¡ÆC11
OR LOAD
LOAD      M1351B	// 12.R_3rd 
AND       M1353B	// STEP A¢Ò¡ÆC12
OR LOAD
LOAD      M1351C	// 13.R_3rd ROT Z 1st
AND       M1353C	// STEP A¢Ò¡ÆC13
OR LOAD
LOAD      M1351D	// 14.R_3rd ALIGN CENTER SUB BW
AND       M1353D	// STEP A¢Ò¡ÆC14
OR LOAD
LOAD      M1351E	// 15.R_3rd ALIGN CENTER BW
AND       M1353E	// STEP A¢Ò¡ÆC15
OR LOAD
LOAD      M1351F	// 16.
AND       M1353F	// STEP A¢Ò¡ÆC16
OR LOAD
LOAD      M13520	// 17.
AND       M13540	// STEP A¢Ò¡ÆC17
OR LOAD
LOAD      M13521	// 18.
AND       M13541	// STEP A¢Ò¡ÆC18
OR LOAD
LOAD      M13522	// 19.
AND       M13542	// STEP A¢Ò¡ÆC19
OR LOAD
LOAD      M13523	// -
AND       M13543	// STEP A¢Ò¡ÆC20
OR LOAD
LOAD      M13524	// -
AND       M13544	// STEP A¢Ò¡ÆC21
OR LOAD
LOAD      M13525	// -
AND       M13545	// STEP A¢Ò¡ÆC22
OR LOAD
LOAD      M13526	// -
AND       M13546	// STEP A¢Ò¡ÆC23
OR LOAD
LOAD      M13527	// -
AND       M13547	// STEP A¢Ò¡ÆC24
OR LOAD
LOAD      M13528	// -
AND       M13548	// STEP A¢Ò¡ÆC25
OR LOAD
LOAD      M13529	// -
AND       M13549	// STEP A¢Ò¡ÆC26
OR LOAD
LOAD      M1352A	// -
AND       M1354A	// STEP A¢Ò¡ÆC27
OR LOAD
LOAD      M1352B	// -
AND       M1354B	// STEP A¢Ò¡ÆC28
OR LOAD
LOAD      M1352C	// -
AND       M1354C	// STEP A¢Ò¡ÆC29
OR LOAD
LOAD      M1352D	// -
AND       M1354D	// STEP A¢Ò¡ÆC35
OR LOAD
LOAD      M1352E	// -
AND       M1354E	// STEP A¢Ò¡ÆC31
OR LOAD
LOAD      M1352F	// 32.R_3rd STEP END
AND       M1354F	// STEP A¢Ò¡ÆC32
OR LOAD
AND LOAD
AND NOT   T1080	// R_3rd MAND STEP DELAY TM
AND       M13580	// R_3rd MAND CYCLE RUN
TON       T1080 D010750	// R_3rd MAND STEP DELAY TM

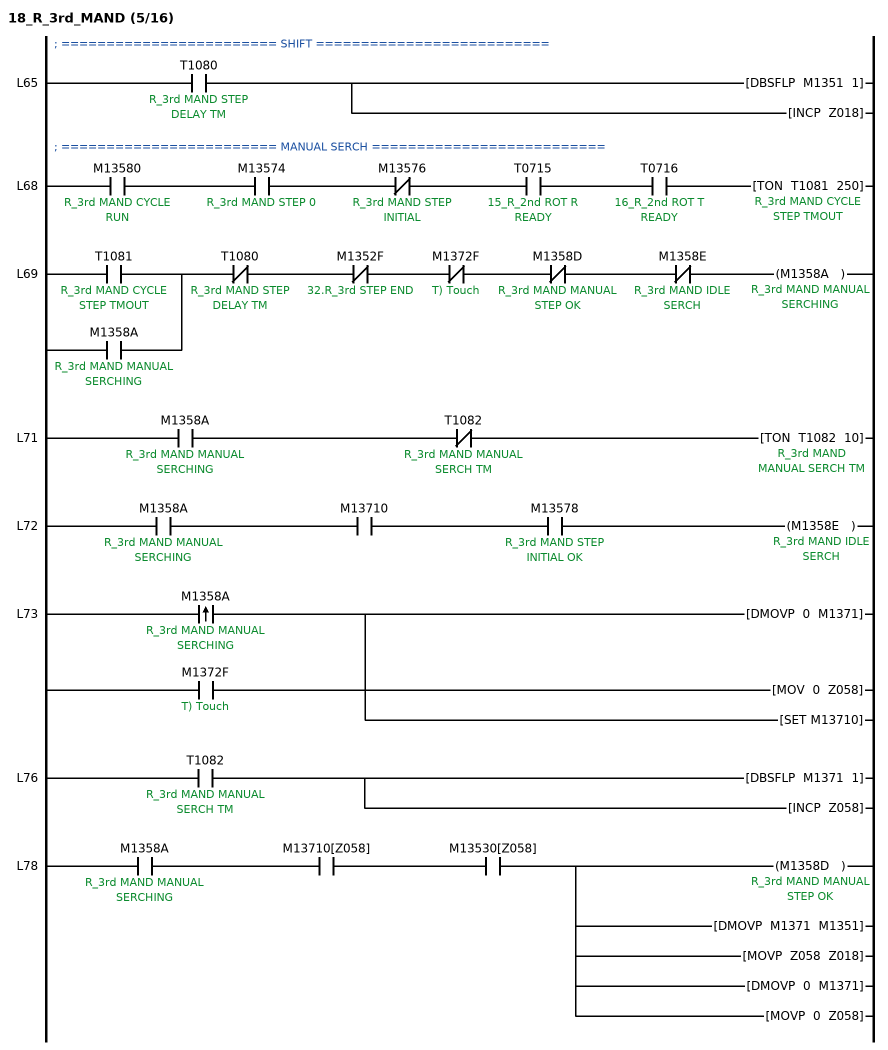
// ======================== SHIFT ==========================
; L65
LOAD      T1080	// R_3rd MAND STEP DELAY TM
DBSFLP    M1351 1
INCP      Z018
// ======================== MANUAL SERCH ==========================
; L68
LOAD      M13580	// R_3rd MAND CYCLE RUN
AND       M13574	// R_3rd MAND STEP 0
AND NOT   M13576	// R_3rd MAND STEP INITIAL
AND       T0715	// 15_R_2nd ROT R READY
AND       T0716	// 16_R_2nd ROT T READY
TON       T1081 250	// R_3rd MAND CYCLE STEP TMOUT
; L69
LOAD      T1081	// R_3rd MAND CYCLE STEP TMOUT
OR        M1358A	// R_3rd MAND MANUAL SERCHING
AND NOT   T1080	// R_3rd MAND STEP DELAY TM
AND NOT   M1352F	// 32.R_3rd STEP END
AND NOT   M1372F	// T) Touch
AND NOT   M1358D	// R_3rd MAND MANUAL STEP OK
AND NOT   M1358E	// R_3rd MAND IDLE SERCH
OUT       M1358A	// R_3rd MAND MANUAL SERCHING
; L71
LOAD      M1358A	// R_3rd MAND MANUAL SERCHING
AND NOT   T1082	// R_3rd MAND MANUAL SERCH TM
TON       T1082 10	// R_3rd MAND MANUAL SERCH TM
; L72
LOAD      M1358A	// R_3rd MAND MANUAL SERCHING
AND       M13710
AND       M13578	// R_3rd MAND STEP INITIAL OK
OUT       M1358E	// R_3rd MAND IDLE SERCH
; L73
LOADP     M1358A	// R_3rd MAND MANUAL SERCHING
OR        M1372F	// T) Touch
DMOVP     0 M1371
MOV       0 Z058
SET       M13710
; L76
LOAD      T1082	// R_3rd MAND MANUAL SERCH TM
DBSFLP    M1371 1
INCP      Z058
; L78
LOAD      M1358A	// R_3rd MAND MANUAL SERCHING
AND       M13710[Z058]
AND       M13530[Z058]
OUT       M1358D	// R_3rd MAND MANUAL STEP OK
DMOVP     M1371 M1351
MOVP      Z058 Z018
DMOVP     0 M1371
MOVP      0 Z058

